  MoveL 3911 to (-68.86, -0.76, -116.32) mm, rotated rx -167.81 ry 3.47 rz -52.11 deg; joints [3.12, -29.463, 100.959, 149.35, 98.482, 24.468, -1.714]
  MoveL 3912 to (-69, -0.7, -116.34) mm, rotated rx -167.81 ry 3.47 rz -52.11 deg; joints [3.124, -29.466, 100.956, 149.354, 98.476, 24.47, -1.714]
  MoveL 3913 to (-69.11, -0.62, -116.37) mm, rotated rx -167.81 ry 3.47 rz -52.11 deg; joints [3.127, -29.469, 100.952, 149.358, 98.47, 24.473, -1.714]
  MoveL 3914 to (-69.19, -0.51, -116.39) mm, rotated rx -167.81 ry 3.47 rz -52.11 deg; joints [3.13, -29.471, 100.946, 149.36, 98.462, 24.477, -1.714]
  MoveL 3915 to (-69.26, -0.38, -116.42) mm, rotated rx -167.81 ry 3.47 rz -52.11 deg; joints [3.131, -29.473, 100.938, 149.362, 98.454, 24.481, -1.714]
  MoveL 3916 to (-69.34, -0.08, -116.48) mm, rotated rx -167.81 ry 3.47 rz -52.11 deg; joints [3.132, -29.476, 100.918, 149.365, 98.435, 24.492, -1.714]
  MoveL 3917 to (-69.29, 0.72, -116.61) mm, rotated rx -167.81 ry 3.47 rz -52.11 deg; joints [3.125, -29.476, 100.864, 149.363, 98.389, 24.522, -1.714]
  MoveL 3918 to (-69.03, 1.69, -116.75) mm, rotated rx -167.81 ry 3.47 rz -52.11 deg; joints [3.11, -29.47, 100.795, 149.353, 98.337, 24.559, -1.714]
  MoveL 3919 to (-68.14, 3.85, -117.02) mm, rotated rx -167.81 ry 3.47 rz -52.11 deg; joints [3.064, -29.451, 100.637, 149.322, 98.225, 24.643, -1.714]
  MoveL 3920 to (-67.07, 6.02, -117.26) mm, rotated rx -167.81 ry 3.47 rz -52.11 deg; joints [3.012, -29.425, 100.475, 149.285, 98.117, 24.728, -1.714]
  MoveL 3921 to (-42.84, 54.26, -122.35) mm, rotated rx -167.81 ry 3.47 rz -52.11 deg; joints [1.884, -28.742, 96.738, 148.461, 95.706, 26.658, -1.714]
  MoveL 3922 to (-41.12, 57.69, -122.71) mm, rotated rx -167.81 ry 3.47 rz -52.11 deg; joints [1.807, -28.687, 96.464, 148.402, 95.535, 26.798, -1.714]
  MoveL 3923 to (-39.28, 60.95, -123.12) mm, rotated rx -167.81 ry 3.47 rz -52.11 deg; joints [1.725, -28.634, 96.204, 148.34, 95.375, 26.934, -1.714]
  MoveL 3924 to (-38.32, 62.09, -123.33) mm, rotated rx -167.81 ry 3.47 rz -52.11 deg; joints [1.685, -28.614, 96.114, 148.307, 95.323, 26.984, -1.714]
  MoveL 3925 to (-37.87, 62.4, -123.43) mm, rotated rx -167.81 ry 3.47 rz -52.11 deg; joints [1.666, -28.607, 96.09, 148.292, 95.312, 26.999, -1.714]
  MoveL 3926 to (-37.65, 62.47, -123.47) mm, rotated rx -167.81 ry 3.47 rz -52.11 deg; joints [1.658, -28.605, 96.085, 148.284, 95.311, 27.004, -1.714]
  MoveL 3927 to (-37.44, 62.47, -123.52) mm, rotated rx -167.81 ry 3.47 rz -52.11 deg; joints [1.65, -28.604, 96.085, 148.277, 95.314, 27.006, -1.714]
  MoveL 3928 to (-37.25, 62.41, -123.55) mm, rotated rx -167.81 ry 3.47 rz -52.11 deg; joints [1.643, -28.603, 96.09, 148.271, 95.32, 27.005, -1.714]
  MoveL 3929 to (-37.06, 62.27, -123.59) mm, rotated rx -167.81 ry 3.47 rz -52.11 deg; joints [1.637, -28.604, 96.102, 148.264, 95.331, 27.001, -1.714]
  MoveL 3930 to (-36.88, 62.06, -123.62) mm, rotated rx -167.81 ry 3.47 rz -52.11 deg; joints [1.631, -28.606, 96.119, 148.258, 95.346, 26.995, -1.714]
  MoveL 3931 to (-36.72, 61.76, -123.64) mm, rotated rx -167.81 ry 3.47 rz -52.11 deg; joints [1.626, -28.609, 96.144, 148.253, 95.365, 26.985, -1.714]
  MoveL 3932 to (-36.22, 59.62, -123.69) mm, rotated rx -167.81 ry 3.47 rz -52.11 deg; joints [1.615, -28.632, 96.317, 148.236, 95.494, 26.909, -1.714]
  MoveL 3933 to (-35.96, 57.54, -123.69) mm, rotated rx -167.81 ry 3.47 rz -52.11 deg; joints [1.614, -28.656, 96.485, 148.227, 95.616, 26.834, -1.714]
  MoveL 3934 to (-35.96, 53.74, -123.74) mm, rotated rx -167.81 ry 3.47 rz -52.11 deg; joints [1.627, -28.711, 96.797, 148.225, 95.833, 26.693, -1.714]
  MoveL 3935 to (-36.73, 50.28, -123.85) mm, rotated rx -167.81 ry 3.47 rz -52.11 deg; joints [1.666, -28.779, 97.091, 148.248, 96.018, 26.561, -1.714]
  MoveL 3936 to (-39.45, 44.87, -124.14) mm, rotated rx -167.81 ry 3.47 rz -52.11 deg; joints [1.779, -28.918, 97.569, 148.33, 96.285, 26.346, -1.714]
  MoveL 3937 to (-40.92, 43.03, -124.27) mm, rotated rx -167.81 ry 3.47 rz -52.11 deg; joints [1.837, -28.977, 97.738, 148.376, 96.367, 26.27, -1.714]
  MoveL 3938 to (-63.78, 16.83, -126.14) mm, rotated rx -167.81 ry 3.47 rz -52.11 deg; joints [2.746, -29.822, 100.106, 149.099, 97.503, 25.201, -1.714]
  MoveL 3939 to (-65.73, 14.58, -126.3) mm, rotated rx -167.81 ry 3.47 rz -52.11 deg; joints [2.825, -29.892, 100.304, 149.161, 97.6, 25.111, -1.714]
  MoveL 3940 to (-67.81, 11.48, -126.54) mm, rotated rx -167.81 ry 3.47 rz -52.11 deg; joints [2.912, -29.978, 100.575, 149.227, 97.744, 24.99, -1.714]
  MoveL 3941 to (-68.34, 10.09, -126.68) mm, rotated rx -167.81 ry 3.47 rz -52.11 deg; joints [2.936, -30.011, 100.694, 149.243, 97.814, 24.939, -1.714]
  MoveL 3942 to (-68.38, 9.55, -126.75) mm, rotated rx -167.81 ry 3.47 rz -52.11 deg; joints [2.939, -30.022, 100.741, 149.243, 97.844, 24.92, -1.714]
  MoveL 3943 to (-68.32, 9.33, -126.79) mm, rotated rx -167.81 ry 3.47 rz -52.11 deg; joints [2.938, -30.025, 100.759, 149.241, 97.857, 24.912, -1.714]
  MoveL 3944 to (-68.22, 9.15, -126.83) mm, rotated rx -167.81 ry 3.47 rz -52.11 deg; joints [2.935, -30.028, 100.775, 149.237, 97.869, 24.906, -1.714]
  MoveL 3945 to (-68.07, 9.01, -126.86) mm, rotated rx -167.81 ry 3.47 rz -52.11 deg; joints [2.929, -30.029, 100.787, 149.231, 97.879, 24.902, -1.714]
  MoveL 3946 to (-67.85, 8.91, -126.9) mm, rotated rx -167.81 ry 3.47 rz -52.11 deg; joints [2.921, -30.028, 100.794, 149.223, 97.888, 24.9, -1.714]
  MoveL 3947 to (-67.58, 8.87, -126.93) mm, rotated rx -167.81 ry 3.47 rz -52.11 deg; joints [2.911, -30.025, 100.798, 149.214, 97.895, 24.9, -1.714]
  MoveL 3948 to (-67.23, 8.88, -126.96) mm, rotated rx -167.81 ry 3.47 rz -52.11 deg; joints [2.898, -30.021, 100.796, 149.202, 97.899, 24.902, -1.714]
  MoveL 3949 to (-65.14, 9.53, -127.09) mm, rotated rx -167.81 ry 3.47 rz -52.11 deg; joints [2.818, -29.984, 100.737, 149.13, 97.894, 24.937, -1.714]
  MoveL 3950 to (-64.67, 9.74, -127.11) mm, rotated rx -167.81 ry 3.47 rz -52.11 deg; joints [2.799, -29.975, 100.719, 149.114, 97.889, 24.947, -1.714]
  MoveL 3951 to (-64.25, 9.95, -127.15) mm, rotated rx -167.81 ry 3.47 rz -52.11 deg; joints [2.783, -29.968, 100.702, 149.1, 97.883, 24.957, -1.714]
  MoveL 3952 to (-63.87, 10.16, -127.23) mm, rotated rx -167.81 ry 3.47 rz -52.11 deg; joints [2.767, -29.964, 100.686, 149.087, 97.876, 24.967, -1.714]
  MoveL 3953 to (-63.48, 10.37, -127.28) mm, rotated rx -167.81 ry 3.47 rz -52.11 deg; joints [2.751, -29.958, 100.671, 149.073, 97.87, 24.977, -1.714]
  MoveL 3954 to (-63.06, 10.57, -127.32) mm, rotated rx -167.81 ry 3.47 rz -52.11 deg; joints [2.735, -29.951, 100.654, 149.059, 97.865, 24.986, -1.714]
  MoveL 3955 to (-58.72, 12.34, -127.33) mm, rotated rx -167.81 ry 3.47 rz -52.11 deg; joints [2.569, -29.854, 100.484, 148.914, 97.831, 25.072, -1.714]
  MoveL 3956 to (-58.31, 12.51, -127.35) mm, rotated rx -167.81 ry 3.47 rz -52.11 deg; joints [2.553, -29.846, 100.468, 148.9, 97.827, 25.08, -1.714]
  MoveL 3957 to (-57.88, 12.7, -127.36) mm, rotated rx -167.81 ry 3.47 rz -52.11 deg; joints [2.536, -29.836, 100.451, 148.886, 97.823, 25.089, -1.714]
  MoveL 3958 to (-56.92, 13.09, -127.36) mm, rotated rx -167.81 ry 3.47 rz -52.11 deg; joints [2.5, -29.815, 100.413, 148.854, 97.816, 25.108, -1.714]
  MoveL 3959 to (-56.39, 13.31, -127.37) mm, rotated rx -167.81 ry 3.47 rz -52.11 deg; joints [2.479, -29.803, 100.392, 148.836, 97.811, 25.119, -1.714]
  MoveL 3960 to (-55.85, 13.57, -127.39) mm, rotated rx -167.81 ry 3.47 rz -52.11 deg; joints [2.458, -29.792, 100.369, 148.818, 97.804, 25.131, -1.714]
  MoveL 3961 to (-55.26, 13.89, -127.42) mm, rotated rx -167.81 ry 3.47 rz -52.11 deg; joints [2.435, -29.78, 100.341, 148.798, 97.795, 25.146, -1.714]
  MoveL 3962 to (-54.72, 14.27, -127.44) mm, rotated rx -167.81 ry 3.47 rz -52.11 deg; joints [2.414, -29.767, 100.309, 148.78, 97.782, 25.163, -1.714]
  MoveL 3963 to (-54.22, 14.69, -127.45) mm, rotated rx -167.81 ry 3.47 rz -52.11 deg; joints [2.394, -29.754, 100.273, 148.764, 97.765, 25.181, -1.714]
  MoveL 3964 to (-55.39, 14.09, -128.43) mm, rotated rx -167.81 ry 3.47 rz -52.11 deg; joints [2.428, -29.845, 100.383, 148.793, 97.776, 25.161, -1.714]
  MoveL 3965 to (-54.92, 15.35, -128.86) mm, rotated rx -167.81 ry 3.47 rz -52.11 deg; joints [2.401, -29.85, 100.305, 148.775, 97.709, 25.212, -1.714]
  MoveL 3966 to (-54.28, 16.69, -129.18) mm, rotated rx -167.81 ry 3.47 rz -52.11 deg; joints [2.368, -29.844, 100.212, 148.751, 97.641, 25.267, -1.714]
  MoveL 3967 to (-53.45, 18.17, -129.41) mm, rotated rx -167.81 ry 3.47 rz -52.11 deg; joints [2.329, -29.828, 100.102, 148.723, 97.568, 25.327, -1.714]
  MoveL 3968 to (-52.29, 19.97, -129.63) mm, rotated rx -167.81 ry 3.47 rz -52.11 deg; joints [2.278, -29.801, 99.964, 148.683, 97.482, 25.4, -1.714]
  MoveL 3969 to (-51.11, 21.74, -129.75) mm, rotated rx -167.81 ry 3.47 rz -52.11 deg; joints [2.226, -29.767, 99.821, 148.645, 97.398, 25.472, -1.714]
  MoveL 3970 to (-49.93, 23.52, -129.86) mm, rotated rx -167.81 ry 3.47 rz -52.11 deg; joints [2.175, -29.732, 99.678, 148.606, 97.314, 25.545, -1.714]
  MoveL 3971 to (-48.77, 25.31, -130.09) mm, rotated rx -167.81 ry 3.47 rz -52.11 deg; joints [2.123, -29.705, 99.54, 148.566, 97.229, 25.618, -1.714]
  MoveL 3972 to (-47.58, 27.08, -130.2) mm, rotated rx -167.81 ry 3.47 rz -52.11 deg; joints [2.072, -29.67, 99.396, 148.527, 97.145, 25.691, -1.714]
  MoveL 3973 to (-46.4, 28.86, -130.44) mm, rotated rx -167.81 ry 3.47 rz -52.11 deg; joints [2.02, -29.643, 99.258, 148.488, 97.061, 25.764, -1.714]
  MoveL 3974 to (-45.21, 30.64, -130.55) mm, rotated rx -167.81 ry 3.47 rz -52.11 deg; joints [1.969, -29.608, 99.114, 148.449, 96.977, 25.837, -1.714]
  MoveL 3975 to (-44.02, 32.41, -130.67) mm, rotated rx -167.81 ry 3.47 rz -52.11 deg; joints [1.918, -29.572, 98.97, 148.41, 96.894, 25.91, -1.714]
  MoveL 3976 to (-42.83, 34.18, -130.91) mm, rotated rx -167.81 ry 3.47 rz -52.11 deg; joints [1.866, -29.544, 98.832, 148.37, 96.81, 25.984, -1.714]
  MoveL 3977 to (-41.68, 35.86, -131.01) mm, rotated rx -167.81 ry 3.47 rz -52.11 deg; joints [1.817, -29.509, 98.693, 148.332, 96.731, 26.053, -1.714]
  MoveL 3978 to (-40.55, 37.5, -131.22) mm, rotated rx -167.81 ry 3.47 rz -52.11 deg; joints [1.768, -29.481, 98.564, 148.294, 96.654, 26.122, -1.714]
  MoveL 3979 to (-39.23, 39.47, -131.38) mm, rotated rx -167.81 ry 3.47 rz -52.11 deg; joints [1.711, -29.443, 98.404, 148.251, 96.561, 26.204, -1.714]
  MoveL 3980 to (-37.68, 41.7, -131.47) mm, rotated rx -167.81 ry 3.47 rz -52.11 deg; joints [1.646, -29.391, 98.215, 148.201, 96.457, 26.296, -1.714]
  MoveL 3981 to (-36.51, 43.42, -131.53) mm, rotated rx -167.81 ry 3.47 rz -52.11 deg; joints [1.598, -29.352, 98.07, 148.164, 96.376, 26.367, -1.714]
  MoveL 3982 to (-35.43, 45.01, -131.66) mm, rotated rx -167.81 ry 3.47 rz -52.11 deg; joints [1.552, -29.32, 97.94, 148.128, 96.301, 26.434, -1.714]
  MoveL 3983 to (-34.31, 46.65, -131.76) mm, rotated rx -167.81 ry 3.47 rz -52.11 deg; joints [1.505, -29.285, 97.803, 148.092, 96.224, 26.502, -1.714]
  MoveL 3984 to (-33.21, 48.26, -131.88) mm, rotated rx -167.81 ry 3.47 rz -52.11 deg; joints [1.459, -29.25, 97.669, 148.056, 96.149, 26.57, -1.714]
  MoveL 3985 to (-32.04, 49.96, -131.95) mm, rotated rx -167.81 ry 3.47 rz -52.11 deg; joints [1.41, -29.211, 97.525, 148.019, 96.069, 26.641, -1.714]
  MoveL 3986 to (-30.78, 51.79, -132.04) mm, rotated rx -167.81 ry 3.47 rz -52.11 deg; joints [1.358, -29.169, 97.37, 147.978, 95.983, 26.718, -1.714]
  MoveL 3987 to (-29.39, 53.75, -132.31) mm, rotated rx -167.81 ry 3.47 rz -52.11 deg; joints [1.299, -29.133, 97.212, 147.932, 95.891, 26.802, -1.714]
  MoveL 3988 to (-28.56, 55.83, -133.29) mm, rotated rx -167.81 ry 3.47 rz -52.11 deg; joints [1.251, -29.152, 97.089, 147.897, 95.781, 26.893, -1.714]
  MoveL 3989 to (-28.58, 54.69, -133.78) mm, rotated rx -167.81 ry 3.47 rz -52.11 deg; joints [1.25, -29.199, 97.209, 147.892, 95.843, 26.854, -1.714]
  MoveL 3990 to (-28.58, 54.09, -134.09) mm, rotated rx -167.81 ry 3.47 rz -52.11 deg; joints [1.249, -29.227, 97.275, 147.889, 95.875, 26.834, -1.714]
  MoveL 3991 to (-28.58, 54, -134.24) mm, rotated rx -167.81 ry 3.47 rz -52.11 deg; joints [1.248, -29.238, 97.291, 147.888, 95.88, 26.832, -1.714]
  MoveL 3992 to (-28.57, 54.34, -134.27) mm, rotated rx -167.81 ry 3.47 rz -52.11 deg; joints [1.246, -29.235, 97.265, 147.887, 95.861, 26.845, -1.714]
  MoveL 3993 to (-28.56, 54.81, -134.29) mm, rotated rx -167.81 ry 3.47 rz -52.11 deg; joints [1.244, -29.23, 97.228, 147.887, 95.834, 26.862, -1.714]
  MoveL 3994 to (-28.54, 55.29, -134.32) mm, rotated rx -167.81 ry 3.47 rz -52.11 deg; joints [1.241, -29.225, 97.19, 147.886, 95.807, 26.881, -1.714]
  MoveL 3995 to (-28.5, 55.74, -134.38) mm, rotated rx -167.81 ry 3.47 rz -52.11 deg; joints [1.237, -29.222, 97.157, 147.885, 95.782, 26.898, -1.714]
  MoveL 3996 to (-28.47, 56.2, -134.43) mm, rotated rx -167.81 ry 3.47 rz -52.11 deg; joints [1.234, -29.218, 97.121, 147.884, 95.756, 26.916, -1.714]
  MoveL 3997 to (-28.46, 56.69, -134.44) mm, rotated rx -167.81 ry 3.47 rz -52.11 deg; joints [1.232, -29.212, 97.082, 147.884, 95.728, 26.934, -1.714]
  MoveL 3998 to (-28.45, 59.31, -134.44) mm, rotated rx -167.81 ry 3.47 rz -52.11 deg; joints [1.223, -29.175, 96.868, 147.885, 95.58, 27.032, -1.714]
  MoveL 3999 to (-28.43, 59.76, -134.46) mm, rotated rx -167.81 ry 3.47 rz -52.11 deg; joints [1.22, -29.17, 96.832, 147.884, 95.554, 27.05, -1.714]
  MoveL 4000 to (-28.4, 60.15, -134.5) mm, rotated rx -167.81 ry 3.47 rz -52.11 deg; joints [1.218, -29.166, 96.802, 147.883, 95.532, 27.064, -1.714]
  MoveL 4001 to (-28.39, 60.61, -134.52) mm, rotated rx -167.81 ry 3.47 rz -52.11 deg; joints [1.215, -29.161, 96.765, 147.883, 95.506, 27.082, -1.714]
  MoveL 4002 to (-28.37, 61.21, -134.54) mm, rotated rx -167.81 ry 3.47 rz -52.11 deg; joints [1.213, -29.153, 96.717, 147.882, 95.473, 27.104, -1.714]
  MoveL 4003 to (-28.33, 61.93, -134.6) mm, rotated rx -167.81 ry 3.47 rz -52.11 deg; joints [1.208, -29.146, 96.66, 147.881, 95.432, 27.132, -1.714]
  MoveL 4004 to (-28.31, 62.55, -134.62) mm, rotated rx -167.81 ry 3.47 rz -52.11 deg; joints [1.205, -29.138, 96.611, 147.88, 95.397, 27.156, -1.714]
  MoveL 4005 to (-28.3, 63.08, -134.63) mm, rotated rx -167.81 ry 3.47 rz -52.11 deg; joints [1.203, -29.131, 96.568, 147.88, 95.367, 27.175, -1.714]
  MoveL 4006 to (-28.29, 64.65, -134.63) mm, rotated rx -167.81 ry 3.47 rz -52.11 deg; joints [1.197, -29.108, 96.438, 147.88, 95.278, 27.234, -1.714]
  MoveL 4007 to (-27.99, 67.55, -134.97) mm, rotated rx -167.81 ry 3.47 rz -52.11 deg; joints [1.173, -29.082, 96.216, 147.868, 95.116, 27.347, -1.714]
  MoveL 4008 to (-27.61, 68.79, -135.4) mm, rotated rx -167.81 ry 3.47 rz -52.11 deg; joints [1.151, -29.084, 96.133, 147.852, 95.049, 27.4, -1.714]
  MoveL 4009 to (-27.09, 69.89, -136) mm, rotated rx -167.81 ry 3.47 rz -52.11 deg; joints [1.122, -29.096, 96.07, 147.83, 94.992, 27.449, -1.714]
  MoveL 4010 to (-25.61, 71.68, -137.71) mm, rotated rx -167.81 ry 3.47 rz -52.11 deg; joints [1.046, -29.15, 96.002, 147.768, 94.904, 27.54, -1.714]
  MoveL 4011 to (-23.55, 72.91, -140.1) mm, rotated rx -167.81 ry 3.47 rz -52.11 deg; joints [0.942, -29.245, 96.011, 147.679, 94.854, 27.62, -1.714]
  MoveL 4012 to (-21.54, 73.36, -142.5) mm, rotated rx -167.81 ry 3.47 rz -52.11 deg; joints [0.844, -29.352, 96.085, 147.593, 94.847, 27.671, -1.714]
  MoveL 4013 to (-20.79, 73.19, -143.44) mm, rotated rx -167.81 ry 3.47 rz -52.11 deg; joints [0.807, -29.4, 96.143, 147.56, 94.863, 27.678, -1.714]
  MoveL 4014 to (-20.22, 72.77, -144.21) mm, rotated rx -167.81 ry 3.47 rz -52.11 deg; joints [0.78, -29.444, 96.214, 147.535, 94.891, 27.673, -1.714]
  MoveL 4015 to (-20, 72.47, -144.53) mm, rotated rx -167.81 ry 3.47 rz -52.11 deg; joints [0.77, -29.465, 96.255, 147.525, 94.91, 27.666, -1.714]
  MoveL 4016 to (-19.82, 72.1, -144.81) mm, rotated rx -167.81 ry 3.47 rz -52.11 deg; joints [0.761, -29.485, 96.299, 147.516, 94.932, 27.655, -1.714]
  MoveL 4017 to (-19.6, 71.17, -145.24) mm, rotated rx -167.81 ry 3.47 rz -52.11 deg; joints [0.752, -29.522, 96.397, 147.505, 94.986, 27.625, -1.714]
  MoveL 4018 to (-19.54, 69.98, -145.49) mm, rotated rx -167.81 ry 3.47 rz -52.11 deg; joints [0.751, -29.555, 96.509, 147.5, 95.053, 27.583, -1.714]
  MoveL 4019 to (-19.67, 68.53, -145.58) mm, rotated rx -167.81 ry 3.47 rz -52.11 deg; joints [0.758, -29.584, 96.634, 147.502, 95.132, 27.529, -1.714]
  MoveL 4020 to (-19.74, 68.01, -145.58) mm, rotated rx -167.81 ry 3.47 rz -52.11 deg; joints [0.762, -29.593, 96.677, 147.504, 95.161, 27.509, -1.714]
  MoveL 4021 to (-19.83, 67.58, -145.52) mm, rotated rx -167.81 ry 3.47 rz -52.11 deg; joints [0.768, -29.597, 96.711, 147.508, 95.184, 27.492, -1.714]
  MoveL 4022 to (-19.93, 67.16, -145.46) mm, rotated rx -167.81 ry 3.47 rz -52.11 deg; joints [0.773, -29.602, 96.743, 147.511, 95.206, 27.474, -1.714]
  MoveL 4023 to (-20.02, 66.69, -145.43) mm, rotated rx -167.81 ry 3.47 rz -52.11 deg; joints [0.778, -29.608, 96.781, 147.514, 95.232, 27.456, -1.714]
  MoveL 4024 to (-20.1, 66.2, -145.41) mm, rotated rx -167.81 ry 3.47 rz -52.11 deg; joints [0.783, -29.615, 96.821, 147.516, 95.258, 27.437, -1.714]
  MoveL 4025 to (-20.17, 65.68, -145.4) mm, rotated rx -167.81 ry 3.47 rz -52.11 deg; joints [0.787, -29.624, 96.865, 147.518, 95.287, 27.417, -1.714]
  MoveL 4026 to (-20.24, 65.16, -145.4) mm, rotated rx -167.81 ry 3.47 rz -52.11 deg; joints [0.791, -29.633, 96.908, 147.52, 95.315, 27.397, -1.714]
  MoveL 4027 to (-20.3, 64.65, -145.42) mm, rotated rx -167.81 ry 3.47 rz -52.11 deg; joints [0.794, -29.642, 96.951, 147.522, 95.343, 27.377, -1.714]
  MoveL 4028 to (-20.35, 64.16, -145.43) mm, rotated rx -167.81 ry 3.47 rz -52.11 deg; joints [0.798, -29.651, 96.993, 147.523, 95.37, 27.359, -1.714]
  MoveL 4029 to (-20.42, 63.7, -145.41) mm, rotated rx -167.81 ry 3.47 rz -52.11 deg; joints [0.802, -29.657, 97.03, 147.525, 95.395, 27.341, -1.714]
  MoveL 4030 to (-20.51, 63.24, -145.37) mm, rotated rx -167.81 ry 3.47 rz -52.11 deg; joints [0.807, -29.663, 97.066, 147.528, 95.42, 27.323, -1.714]
  MoveL 4031 to (-20.61, 62.71, -145.32) mm, rotated rx -167.81 ry 3.47 rz -52.11 deg; joints [0.813, -29.669, 97.108, 147.531, 95.449, 27.301, -1.714]
  MoveL 4032 to (-20.75, 62.02, -145.27) mm, rotated rx -167.81 ry 3.47 rz -52.11 deg; joints [0.82, -29.679, 97.163, 147.536, 95.486, 27.274, -1.714]
  MoveL 4033 to (-20.86, 61.38, -145.24) mm, rotated rx -167.81 ry 3.47 rz -52.11 deg; joints [0.826, -29.688, 97.215, 147.539, 95.52, 27.249, -1.714]
  MoveL 4034 to (-21.2, 58.79, -145.24) mm, rotated rx -167.81 ry 3.47 rz -52.11 deg; joints [0.847, -29.731, 97.431, 147.548, 95.662, 27.15, -1.714]
  MoveL 4035 to (-21.3, 58.17, -145.21) mm, rotated rx -167.81 ry 3.47 rz -52.11 deg; joints [0.853, -29.739, 97.48, 147.551, 95.696, 27.126, -1.714]
  MoveL 4036 to (-21.4, 57.62, -145.15) mm, rotated rx -167.81 ry 3.47 rz -52.11 deg; joints [0.859, -29.745, 97.523, 147.555, 95.725, 27.104, -1.714]
  MoveL 4037 to (-21.44, 57.42, -145) mm, rotated rx -167.81 ry 3.47 rz -52.11 deg; joints [0.862, -29.739, 97.532, 147.557, 95.737, 27.095, -1.714]
  MoveL 4038 to (-21.42, 57.54, -144.73) mm, rotated rx -167.81 ry 3.47 rz -52.11 deg; joints [0.864, -29.72, 97.507, 147.559, 95.732, 27.097, -1.714]
  MoveL 4039 to (-21.33, 57.99, -144.33) mm, rotated rx -167.81 ry 3.47 rz -52.11 deg; joints [0.864, -29.687, 97.448, 147.56, 95.71, 27.111, -1.714]
  MoveL 4040 to (-22.34, 57.8, -143.53) mm, rotated rx -167.81 ry 3.47 rz -52.11 deg; joints [0.91, -29.658, 97.43, 147.601, 95.71, 27.09, -1.714]
  MoveL 4041 to (-23.69, 56.35, -143.31) mm, rotated rx -167.81 ry 3.47 rz -52.11 deg; joints [0.965, -29.689, 97.549, 147.645, 95.773, 27.025, -1.714]
  MoveL 4042 to (-25.04, 54.87, -143.15) mm, rotated rx -167.81 ry 3.47 rz -52.11 deg; joints [1.019, -29.725, 97.674, 147.689, 95.838, 26.96, -1.714]
  MoveL 4043 to (-26.42, 53.34, -143) mm, rotated rx -167.81 ry 3.47 rz -52.11 deg; joints [1.075, -29.762, 97.803, 147.734, 95.905, 26.893, -1.714]
  MoveL 4044 to (-27.69, 51.96, -142.71) mm, rotated rx -167.81 ry 3.47 rz -52.11 deg; joints [1.128, -29.786, 97.912, 147.777, 95.966, 26.83, -1.714]
  MoveL 4045 to (-29.11, 50.39, -142.52) mm, rotated rx -167.81 ry 3.47 rz -52.11 deg; joints [1.186, -29.821, 98.042, 147.823, 96.034, 26.761, -1.714]
  MoveL 4046 to (-30.59, 48.75, -142.33) mm, rotated rx -167.81 ry 3.47 rz -52.11 deg; joints [1.247, -29.859, 98.179, 147.872, 96.106, 26.689, -1.714]
  MoveL 4047 to (-32.09, 47.08, -142.25) mm, rotated rx -167.81 ry 3.47 rz -52.11 deg; joints [1.307, -29.903, 98.323, 147.92, 96.179, 26.617, -1.714]
  MoveL 4048 to (-33.9, 45.04, -142.16) mm, rotated rx -167.81 ry 3.47 rz -52.11 deg; joints [1.38, -29.958, 98.499, 147.979, 96.268, 26.529, -1.714]
  MoveL 4049 to (-35.2, 43.57, -142.05) mm, rotated rx -167.81 ry 3.47 rz -52.11 deg; joints [1.433, -29.994, 98.623, 148.021, 96.332, 26.466, -1.714]
  MoveL 4050 to (-36.41, 42.2, -141.83) mm, rotated rx -167.81 ry 3.47 rz -52.11 deg; joints [1.483, -30.021, 98.732, 148.061, 96.392, 26.406, -1.714]
  MoveL 4051 to (-37.75, 40.69, -141.64) mm, rotated rx -167.81 ry 3.47 rz -52.11 deg; joints [1.539, -30.053, 98.855, 148.106, 96.459, 26.341, -1.714]
  MoveL 4052 to (-39.16, 39.09, -141.52) mm, rotated rx -167.81 ry 3.47 rz -52.11 deg; joints [1.597, -30.091, 98.99, 148.152, 96.529, 26.272, -1.714]
  MoveL 4053 to (-40.55, 37.5, -141.35) mm, rotated rx -167.81 ry 3.47 rz -52.11 deg; joints [1.654, -30.126, 99.12, 148.198, 96.6, 26.204, -1.714]
  MoveL 4054 to (-41.94, 35.91, -141.23) mm, rotated rx -167.81 ry 3.47 rz -52.11 deg; joints [1.712, -30.163, 99.252, 148.244, 96.669, 26.136, -1.714]
  MoveL 4055 to (-43.37, 34.26, -141.05) mm, rotated rx -167.81 ry 3.47 rz -52.11 deg; joints [1.771, -30.199, 99.386, 148.291, 96.742, 26.066, -1.714]
  MoveL 4056 to (-44.77, 32.65, -140.93) mm, rotated rx -167.81 ry 3.47 rz -52.11 deg; joints [1.829, -30.236, 99.519, 148.337, 96.813, 25.997, -1.714]
  MoveL 4057 to (-46.15, 31.03, -140.7) mm, rotated rx -167.81 ry 3.47 rz -52.11 deg; joints [1.888, -30.267, 99.648, 148.384, 96.885, 25.928, -1.714]
  MoveL 4058 to (-47.55, 29.41, -140.58) mm, rotated rx -167.81 ry 3.47 rz -52.11 deg; joints [1.946, -30.305, 99.781, 148.43, 96.956, 25.86, -1.714]
  MoveL 4059 to (-48.94, 27.8, -140.47) mm, rotated rx -167.81 ry 3.47 rz -52.11 deg; joints [2.004, -30.342, 99.914, 148.476, 97.027, 25.792, -1.714]
  MoveL 4060 to (-50.32, 26.16, -140.24) mm, rotated rx -167.81 ry 3.47 rz -52.11 deg; joints [2.063, -30.372, 100.043, 148.523, 97.1, 25.722, -1.714]
  MoveL 4061 to (-51.53, 24.65, -140.04) mm, rotated rx -167.81 ry 3.47 rz -52.11 deg; joints [2.115, -30.399, 100.161, 148.564, 97.168, 25.659, -1.714]
  MoveL 4062 to (-52.58, 23.23, -139.75) mm, rotated rx -167.81 ry 3.47 rz -52.11 deg; joints [2.162, -30.416, 100.265, 148.6, 97.234, 25.599, -1.714]
  MoveL 4063 to (-53.49, 21.88, -139.34) mm, rotated rx -167.81 ry 3.47 rz -52.11 deg; joints [2.205, -30.422, 100.357, 148.633, 97.3, 25.541, -1.714]
  MoveL 4064 to (-52.18, 22.58, -138.42) mm, rotated rx -167.81 ry 3.47 rz -52.11 deg; joints [2.165, -30.331, 100.241, 148.599, 97.286, 25.566, -1.714]
  MoveL 4065 to (-52.64, 22.23, -138.41) mm, rotated rx -167.81 ry 3.47 rz -52.11 deg; joints [2.183, -30.343, 100.271, 148.614, 97.298, 25.551, -1.714]
  MoveL 4066 to (-53.09, 21.94, -138.38) mm, rotated rx -167.81 ry 3.47 rz -52.11 deg; joints [2.201, -30.353, 100.296, 148.629, 97.308, 25.538, -1.714]
  MoveL 4067 to (-53.5, 21.72, -138.32) mm, rotated rx -167.81 ry 3.47 rz -52.11 deg; joints [2.217, -30.359, 100.313, 148.643, 97.314, 25.527, -1.714]
  MoveL 4068 to (-53.91, 21.54, -138.26) mm, rotated rx -167.81 ry 3.47 rz -52.11 deg; joints [2.234, -30.364, 100.328, 148.657, 97.319, 25.518, -1.714]
  MoveL 4069 to (-54.34, 21.38, -138.21) mm, rotated rx -167.81 ry 3.47 rz -52.11 deg; joints [2.251, -30.371, 100.341, 148.672, 97.322, 25.509, -1.714]
  MoveL 4070 to (-54.81, 21.23, -138.17) mm, rotated rx -167.81 ry 3.47 rz -52.11 deg; joints [2.268, -30.379, 100.355, 148.688, 97.324, 25.501, -1.714]
  MoveL 4071 to (-55.31, 21.08, -138.16) mm, rotated rx -167.81 ry 3.47 rz -52.11 deg; joints [2.288, -30.389, 100.369, 148.705, 97.324, 25.493, -1.714]
  MoveL 4072 to (-55.82, 20.95, -138.16) mm, rotated rx -167.81 ry 3.47 rz -52.11 deg; joints [2.307, -30.4, 100.384, 148.722, 97.324, 25.486, -1.714]
  MoveL 4073 to (-56.27, 20.82, -138.15) mm, rotated rx -167.81 ry 3.47 rz -52.11 deg; joints [2.324, -30.409, 100.397, 148.737, 97.324, 25.478, -1.714]
  MoveL 4074 to (-56.67, 20.69, -138.12) mm, rotated rx -167.81 ry 3.47 rz -52.11 deg; joints [2.339, -30.416, 100.409, 148.75, 97.326, 25.471, -1.714]
  MoveL 4075 to (-57.14, 20.55, -138.11) mm, rotated rx -167.81 ry 3.47 rz -52.11 deg; joints [2.357, -30.425, 100.422, 148.766, 97.326, 25.464, -1.714]
  MoveL 4076 to (-57.64, 20.42, -138.11) mm, rotated rx -167.81 ry 3.47 rz -52.11 deg; joints [2.375, -30.436, 100.437, 148.783, 97.326, 25.457, -1.714]
  MoveL 4077 to (-58.23, 20.25, -138.09) mm, rotated rx -167.81 ry 3.47 rz -52.11 deg; joints [2.398, -30.447, 100.453, 148.803, 97.327, 25.447, -1.714]
  MoveL 4078 to (-58.9, 20.05, -138.04) mm, rotated rx -167.81 ry 3.47 rz -52.11 deg; joints [2.423, -30.459, 100.471, 148.825, 97.328, 25.436, -1.714]
  MoveL 4079 to (-59.48, 19.89, -138.02) mm, rotated rx -167.81 ry 3.47 rz -52.11 deg; joints [2.445, -30.47, 100.488, 148.845, 97.328, 25.427, -1.714]
  MoveL 4080 to (-60.1, 19.71, -138) mm, rotated rx -167.81 ry 3.47 rz -52.11 deg; joints [2.469, -30.482, 100.505, 148.865, 97.329, 25.417, -1.714]
  MoveL 4081 to (-60.78, 19.49, -137.96) mm, rotated rx -167.81 ry 3.47 rz -52.11 deg; joints [2.495, -30.494, 100.525, 148.888, 97.331, 25.406, -1.714]
  MoveL 4082 to (-61.34, 19.33, -137.95) mm, rotated rx -167.81 ry 3.47 rz -52.11 deg; joints [2.516, -30.505, 100.541, 148.907, 97.331, 25.397, -1.714]
  MoveL 4083 to (-61.87, 19.19, -137.94) mm, rotated rx -167.81 ry 3.47 rz -52.11 deg; joints [2.536, -30.516, 100.556, 148.925, 97.331, 25.389, -1.714]
  MoveL 4084 to (-63.39, 18.79, -137.94) mm, rotated rx -167.81 ry 3.47 rz -52.11 deg; joints [2.593, -30.548, 100.599, 148.976, 97.33, 25.367, -1.714]
  MoveL 4085 to (-64.81, 18.49, -138.03) mm, rotated rx -167.81 ry 3.47 rz -52.11 deg; joints [2.645, -30.583, 100.637, 149.022, 97.324, 25.349, -1.714]
  MoveL 4086 to (-65.99, 18.39, -138.28) mm, rotated rx -167.81 ry 3.47 rz -52.11 deg; joints [2.686, -30.622, 100.667, 149.06, 97.31, 25.342, -1.714]
  MoveL 4087 to (-66.95, 18.5, -138.7) mm, rotated rx -167.81 ry 3.47 rz -52.11 deg; joints [2.715, -30.665, 100.689, 149.088, 97.286, 25.344, -1.714]
  MoveL 4088 to (-67.33, 18.63, -138.98) mm, rotated rx -167.81 ry 3.47 rz -52.11 deg; joints [2.726, -30.688, 100.696, 149.098, 97.271, 25.349, -1.714]
  MoveL 4089 to (-67.66, 18.81, -139.29) mm, rotated rx -167.81 ry 3.47 rz -52.11 deg; joints [2.733, -30.712, 100.702, 149.106, 97.253, 25.357, -1.714]
  MoveL 4090 to (-68.15, 19.32, -140.05) mm, rotated rx -167.81 ry 3.47 rz -52.11 deg; joints [2.74, -30.764, 100.706, 149.116, 97.212, 25.379, -1.714]
  MoveL 4091 to (-68.4, 20.04, -140.98) mm, rotated rx -167.81 ry 3.47 rz -52.11 deg; joints [2.736, -30.819, 100.702, 149.116, 97.161, 25.411, -1.714]
  MoveL 4092 to (-68.2, 22.08, -143.34) mm, rotated rx -167.81 ry 3.47 rz -52.11 deg; joints [2.694, -30.943, 100.668, 149.088, 97.033, 25.506, -1.714]
  MoveL 4093 to (-67.23, 24.28, -145.71) mm, rotated rx -167.81 ry 3.47 rz -52.11 deg; joints [2.623, -31.051, 100.615, 149.034, 96.908, 25.61, -1.714]
  MoveL 4094 to (-65.63, 25.97, -147.39) mm, rotated rx -167.81 ry 3.47 rz -52.11 deg; joints [2.539, -31.11, 100.562, 148.965, 96.827, 25.694, -1.714]
  MoveL 4095 to (-64.6, 26.62, -147.98) mm, rotated rx -167.81 ry 3.47 rz -52.11 deg; joints [2.492, -31.122, 100.535, 148.925, 96.802, 25.728, -1.714]
  MoveL 4096 to (-63.41, 27.14, -148.41) mm, rotated rx -167.81 ry 3.47 rz -52.11 deg; joints [2.442, -31.121, 100.507, 148.882, 96.789, 25.757, -1.714]
  MoveL 4097 to (-60.57, 27.81, -148.74) mm, rotated rx -167.81 ry 3.47 rz -52.11 deg; joints [2.333, -31.083, 100.452, 148.785, 96.794, 25.799, -1.714]
  MoveL 4098 to (-56.42, 28.35, -148.74) mm, rotated rx -167.81 ry 3.47 rz -52.11 deg; joints [2.18, -31, 100.378, 148.647, 96.829, 25.841, -1.714]
  MoveL 4099 to (-55.88, 28.43, -148.76) mm, rotated rx -167.81 ry 3.47 rz -52.11 deg; joints [2.16, -30.991, 100.368, 148.629, 96.832, 25.847, -1.714]
  MoveL 4100 to (-55.36, 28.53, -148.8) mm, rotated rx -167.81 ry 3.47 rz -52.11 deg; joints [2.14, -30.983, 100.359, 148.611, 96.835, 25.854, -1.714]
  MoveL 4101 to (-54.84, 28.64, -148.86) mm, rotated rx -167.81 ry 3.47 rz -52.11 deg; joints [2.12, -30.976, 100.349, 148.593, 96.836, 25.861, -1.714]
  MoveL 4102 to (-54.34, 28.76, -148.95) mm, rotated rx -167.81 ry 3.47 rz -52.11 deg; joints [2.101, -30.97, 100.34, 148.576, 96.836, 25.869, -1.714]
  MoveL 4103 to (-53.84, 28.88, -149.02) mm, rotated rx -167.81 ry 3.47 rz -52.11 deg; joints [2.081, -30.965, 100.331, 148.559, 96.837, 25.877, -1.714]
  MoveL 4104 to (-53.37, 28.97, -149.06) mm, rotated rx -167.81 ry 3.47 rz -52.11 deg; joints [2.063, -30.958, 100.322, 148.543, 96.839, 25.883, -1.714]
  MoveL 4105 to (-52.89, 29.04, -149.08) mm, rotated rx -167.81 ry 3.47 rz -52.11 deg; joints [2.046, -30.949, 100.314, 148.527, 96.842, 25.889, -1.714]
  MoveL 4106 to (-52.37, 29.11, -149.08) mm, rotated rx -167.81 ry 3.47 rz -52.11 deg; joints [2.027, -30.939, 100.304, 148.509, 96.846, 25.894, -1.714]
  MoveL 4107 to (-51.75, 29.21, -149.11) mm, rotated rx -167.81 ry 3.47 rz -52.11 deg; joints [2.003, -30.928, 100.293, 148.489, 96.85, 25.901, -1.714]
  MoveL 4108 to (-51.08, 29.34, -149.17) mm, rotated rx -167.81 ry 3.47 rz -52.11 deg; joints [1.978, -30.918, 100.281, 148.466, 96.853, 25.91, -1.714]
  MoveL 4109 to (-50.5, 29.45, -149.19) mm, rotated rx -167.81 ry 3.47 rz -52.11 deg; joints [1.956, -30.907, 100.268, 148.446, 96.855, 25.918, -1.714]
  MoveL 4110 to (-49.96, 29.6, -149.2) mm, rotated rx -167.81 ry 3.47 rz -52.11 deg; joints [1.936, -30.896, 100.253, 148.429, 96.855, 25.926, -1.714]
  MoveL 4111 to (-49.44, 29.79, -149.21) mm, rotated rx -167.81 ry 3.47 rz -52.11 deg; joints [1.916, -30.885, 100.233, 148.412, 96.853, 25.936, -1.714]
  MoveL 4112 to (-48.96, 30.1, -149.21) mm, rotated rx -167.81 ry 3.47 rz -52.11 deg; joints [1.898, -30.872, 100.205, 148.396, 96.843, 25.95, -1.714]
  MoveL 4113 to (-48.48, 30.48, -149.21) mm, rotated rx -167.81 ry 3.47 rz -52.11 deg; joints [1.879, -30.859, 100.171, 148.38, 96.828, 25.967, -1.714]
  MoveL 4114 to (-49.9, 29.8, -150.16) mm, rotated rx -167.81 ry 3.47 rz -52.11 deg; joints [1.922, -30.954, 100.288, 148.418, 96.839, 25.942, -1.714]
  MoveL 4115 to (-49.13, 30.78, -150.59) mm, rotated rx -167.81 ry 3.47 rz -52.11 deg; joints [1.886, -30.955, 100.227, 148.389, 96.793, 25.986, -1.714]
  MoveL 4116 to (-48.17, 31.82, -150.91) mm, rotated rx -167.81 ry 3.47 rz -52.11 deg; joints [1.844, -30.945, 100.153, 148.355, 96.746, 26.033, -1.714]
  MoveL 4117 to (-47.03, 32.96, -151.16) mm, rotated rx -167.81 ry 3.47 rz -52.11 deg; joints [1.795, -30.926, 100.067, 148.315, 96.698, 26.083, -1.714]
  MoveL 4118 to (-45.45, 34.38, -151.27) mm, rotated rx -167.81 ry 3.47 rz -52.11 deg; joints [1.731, -30.887, 99.947, 148.263, 96.641, 26.145, -1.714]
  MoveL 4119 to (-43.87, 35.82, -151.5) mm, rotated rx -167.81 ry 3.47 rz -52.11 deg; joints [1.666, -30.854, 99.831, 148.21, 96.583, 26.209, -1.714]
  MoveL 4120 to (-42.28, 37.24, -151.62) mm, rotated rx -167.81 ry 3.47 rz -52.11 deg; joints [1.603, -30.814, 99.711, 148.157, 96.526, 26.271, -1.714]
  MoveL 4121 to (-40.69, 38.65, -151.74) mm, rotated rx -167.81 ry 3.47 rz -52.11 deg; joints [1.539, -30.774, 99.59, 148.105, 96.47, 26.334, -1.714]
  MoveL 4122 to (-39.1, 40.08, -151.97) mm, rotated rx -167.81 ry 3.47 rz -52.11 deg; joints [1.474, -30.742, 99.474, 148.051, 96.412, 26.398, -1.714]
  MoveL 4123 to (-37.5, 41.49, -152.09) mm, rotated rx -167.81 ry 3.47 rz -52.11 deg; joints [1.41, -30.702, 99.353, 147.999, 96.356, 26.461, -1.714]
  MoveL 4124 to (-35.9, 42.9, -152.21) mm, rotated rx -167.81 ry 3.47 rz -52.11 deg; joints [1.346, -30.661, 99.232, 147.947, 96.3, 26.524, -1.714]
  MoveL 4125 to (-34.06, 44.53, -152.37) mm, rotated rx -167.81 ry 3.47 rz -52.11 deg; joints [1.273, -30.616, 99.093, 147.886, 96.234, 26.597, -1.714]
  MoveL 4126 to (-32.48, 45.92, -152.56) mm, rotated rx -167.81 ry 3.47 rz -52.11 deg; joints [1.209, -30.581, 98.978, 147.834, 96.179, 26.66, -1.714]
  MoveL 4127 to (-30.75, 47.44, -152.76) mm, rotated rx -167.81 ry 3.47 rz -52.11 deg; joints [1.139, -30.541, 98.849, 147.776, 96.118, 26.729, -1.714]
  MoveL 4128 to (-29.04, 48.92, -153.01) mm, rotated rx -167.81 ry 3.47 rz -52.11 deg; joints [1.071, -30.505, 98.727, 147.72, 96.058, 26.797, -1.714]
  MoveL 4129 to (-27.43, 50.33, -153.14) mm, rotated rx -167.81 ry 3.47 rz -52.11 deg; joints [1.007, -30.464, 98.605, 147.667, 96.003, 26.861, -1.714]
  MoveL 4130 to (-25.83, 51.73, -153.14) mm, rotated rx -167.81 ry 3.47 rz -52.11 deg; joints [0.945, -30.415, 98.476, 147.616, 95.947, 26.923, -1.714]
  MoveL 4131 to (-24.24, 53.11, -153.21) mm, rotated rx -167.81 ry 3.47 rz -52.11 deg; joints [0.883, -30.371, 98.353, 147.565, 95.893, 26.986, -1.714]
  MoveL 4132 to (-22.67, 54.45, -153.43) mm, rotated rx -167.81 ry 3.47 rz -52.11 deg; joints [0.82, -30.337, 98.241, 147.514, 95.84, 27.048, -1.714]
  MoveL 4133 to (-20.9, 55.92, -153.78) mm, rotated rx -167.81 ry 3.47 rz -52.11 deg; joints [0.749, -30.305, 98.122, 147.454, 95.781, 27.118, -1.714]
  MoveL 4134 to (-19.51, 57.08, -153.99) mm, rotated rx -167.81 ry 3.47 rz -52.11 deg; joints [0.693, -30.276, 98.025, 147.409, 95.735, 27.172, -1.714]
  MoveL 4135 to (-17.61, 58.64, -154.29) mm, rotated rx -167.81 ry 3.47 rz -52.11 deg; joints [0.618, -30.238, 97.895, 147.346, 95.673, 27.246, -1.714]
  MoveL 4136 to (-15.93, 60.07, -154.39) mm, rotated rx -167.81 ry 3.47 rz -52.11 deg; joints [0.553, -30.192, 97.767, 147.292, 95.617, 27.312, -1.714]
  MoveL 4137 to (-14.33, 61.47, -154.41) mm, rotated rx -167.81 ry 3.47 rz -52.11 deg; joints [0.491, -30.143, 97.637, 147.242, 95.561, 27.376, -1.714]
  MoveL 4138 to (-13.45, 61.58, -155.19) mm, rotated rx -167.81 ry 3.47 rz -52.11 deg; joints [0.451, -30.174, 97.66, 147.206, 95.564, 27.393, -1.714]
  MoveL 4139 to (-13.64, 61.18, -155.59) mm, rotated rx -167.81 ry 3.47 rz -52.11 deg; joints [0.454, -30.208, 97.716, 147.208, 95.581, 27.38, -1.714]
  MoveL 4140 to (-13.71, 61.06, -155.83) mm, rotated rx -167.81 ry 3.47 rz -52.11 deg; joints [0.454, -30.227, 97.74, 147.208, 95.585, 27.377, -1.714]
  MoveL 4141 to (-13.67, 61.2, -155.95) mm, rotated rx -167.81 ry 3.47 rz -52.11 deg; joints [0.451, -30.232, 97.735, 147.205, 95.577, 27.384, -1.714]
  MoveL 4142 to (-13.55, 61.57, -155.98) mm, rotated rx -167.81 ry 3.47 rz -52.11 deg; joints [0.445, -30.226, 97.704, 147.202, 95.558, 27.399, -1.714]
  MoveL 4143 to (-13.42, 62.02, -155.98) mm, rotated rx -167.81 ry 3.47 rz -52.11 deg; joints [0.44, -30.217, 97.666, 147.198, 95.534, 27.417, -1.714]
  MoveL 4144 to (-13.02, 63.54, -155.98) mm, rotated rx -167.81 ry 3.47 rz -52.11 deg; joints [0.421, -30.188, 97.537, 147.186, 95.455, 27.477, -1.714]
  MoveL 4145 to (-12.86, 64.07, -156) mm, rotated rx -167.81 ry 3.47 rz -52.11 deg; joints [0.413, -30.178, 97.493, 147.182, 95.427, 27.498, -1.714]
  MoveL 4146 to (-12.69, 64.6, -156.05) mm, rotated rx -167.81 ry 3.47 rz -52.11 deg; joints [0.405, -30.171, 97.451, 147.176, 95.4, 27.52, -1.714]
  MoveL 4147 to (-12.49, 65.13, -156.13) mm, rotated rx -167.81 ry 3.47 rz -52.11 deg; joints [0.396, -30.164, 97.409, 147.169, 95.372, 27.542, -1.714]
  MoveL 4148 to (-12.31, 65.66, -156.19) mm, rotated rx -167.81 ry 3.47 rz -52.11 deg; joints [0.387, -30.157, 97.367, 147.163, 95.345, 27.564, -1.714]
  MoveL 4149 to (-12.15, 66.17, -156.22) mm, rotated rx -167.81 ry 3.47 rz -52.11 deg; joints [0.38, -30.148, 97.325, 147.159, 95.319, 27.584, -1.714]
  MoveL 4150 to (-12.01, 66.64, -156.24) mm, rotated rx -167.81 ry 3.47 rz -52.11 deg; joints [0.373, -30.14, 97.286, 147.154, 95.294, 27.603, -1.714]
  MoveL 4151 to (-11.86, 67.08, -156.28) mm, rotated rx -167.81 ry 3.47 rz -52.11 deg; joints [0.366, -30.133, 97.251, 147.15, 95.271, 27.621, -1.714]
  MoveL 4152 to (-11.72, 67.49, -156.32) mm, rotated rx -167.81 ry 3.47 rz -52.11 deg; joints [0.36, -30.127, 97.217, 147.145, 95.25, 27.638, -1.714]
  MoveL 4153 to (-11.58, 67.97, -156.33) mm, rotated rx -167.81 ry 3.47 rz -52.11 deg; joints [0.353, -30.118, 97.177, 147.141, 95.225, 27.658, -1.714]
  MoveL 4154 to (-11.42, 68.53, -156.35) mm, rotated rx -167.81 ry 3.47 rz -52.11 deg; joints [0.346, -30.108, 97.13, 147.136, 95.195, 27.68, -1.714]
  MoveL 4155 to (-11.2, 69.2, -156.41) mm, rotated rx -167.81 ry 3.47 rz -52.11 deg; joints [0.335, -30.097, 97.076, 147.129, 95.161, 27.707, -1.714]
  MoveL 4156 to (-11.02, 69.78, -156.43) mm, rotated rx -167.81 ry 3.47 rz -52.11 deg; joints [0.327, -30.087, 97.027, 147.123, 95.131, 27.731, -1.714]
  MoveL 4157 to (-10.47, 71.81, -156.44) mm, rotated rx -167.81 ry 3.47 rz -52.11 deg; joints [0.302, -30.047, 96.854, 147.108, 95.024, 27.812, -1.714]
  MoveL 4158 to (-9.45, 74.54, -156.77) mm, rotated rx -167.81 ry 3.47 rz -52.11 deg; joints [0.255, -30.007, 96.635, 147.074, 94.884, 27.925, -1.714]
  MoveL 4159 to (-8.78, 75.64, -157.18) mm, rotated rx -167.81 ry 3.47 rz -52.11 deg; joints [0.223, -30.003, 96.558, 147.049, 94.829, 27.976, -1.714]
  MoveL 4160 to (-8, 76.58, -157.76) mm, rotated rx -167.81 ry 3.47 rz -52.11 deg; joints [0.187, -30.01, 96.502, 147.02, 94.785, 28.022, -1.714]
  MoveL 4161 to (-6.14, 77.94, -159.41) mm, rotated rx -167.81 ry 3.47 rz -52.11 deg; joints [0.099, -30.057, 96.457, 146.946, 94.726, 28.102, -1.714]
  MoveL 4162 to (-3.86, 78.62, -161.71) mm, rotated rx -167.81 ry 3.47 rz -52.11 deg; joints [-0.009, -30.148, 96.499, 146.852, 94.709, 28.166, -1.714]
  MoveL 4163 to (-1.84, 78.54, -164.02) mm, rotated rx -167.81 ry 3.47 rz -52.11 deg; joints [-0.106, -30.256, 96.605, 146.766, 94.729, 28.199, -1.714]
  MoveL 4164 to (-1.17, 78.2, -164.93) mm, rotated rx -167.81 ry 3.47 rz -52.11 deg; joints [-0.139, -30.305, 96.674, 146.736, 94.753, 28.199, -1.714]
  MoveL 4165 to (-0.73, 77.65, -165.67) mm, rotated rx -167.81 ry 3.47 rz -52.11 deg; joints [-0.162, -30.352, 96.754, 146.714, 94.785, 28.189, -1.714]
  MoveL 4166 to (-0.6, 77.3, -165.98) mm, rotated rx -167.81 ry 3.47 rz -52.11 deg; joints [-0.169, -30.374, 96.798, 146.707, 94.805, 28.179, -1.714]
  MoveL 4167 to (-0.53, 76.9, -166.24) mm, rotated rx -167.81 ry 3.47 rz -52.11 deg; joints [-0.173, -30.396, 96.845, 146.702, 94.827, 28.167, -1.714]
  MoveL 4168 to (-0.56, 75.94, -166.66) mm, rotated rx -167.81 ry 3.47 rz -52.11 deg; joints [-0.175, -30.437, 96.946, 146.698, 94.878, 28.134, -1.714]
  MoveL 4169 to (-0.81, 74.78, -166.9) mm, rotated rx -167.81 ry 3.47 rz -52.11 deg; joints [-0.166, -30.476, 97.059, 146.702, 94.938, 28.09, -1.714]
  MoveL 4170 to (-1.3, 73.42, -166.99) mm, rotated rx -167.81 ry 3.47 rz -52.11 deg; joints [-0.146, -30.511, 97.182, 146.716, 95.007, 28.035, -1.714]
  MoveL 4171 to (-2.69, 70.03, -166.99) mm, rotated rx -167.81 ry 3.47 rz -52.11 deg; joints [-0.088, -30.589, 97.477, 146.756, 95.176, 27.896, -1.714]
  MoveL 4172 to (-2.88, 69.6, -166.97) mm, rotated rx -167.81 ry 3.47 rz -52.11 deg; joints [-0.08, -30.598, 97.513, 146.762, 95.197, 27.878, -1.714]
  MoveL 4173 to (-3.05, 69.23, -166.94) mm, rotated rx -167.81 ry 3.47 rz -52.11 deg; joints [-0.073, -30.605, 97.545, 146.767, 95.216, 27.863, -1.714]
  MoveL 4174 to (-3.24, 68.8, -166.93) mm, rotated rx -167.81 ry 3.47 rz -52.11 deg; joints [-0.065, -30.614, 97.582, 146.773, 95.237, 27.845, -1.714]
  MoveL 4175 to (-4.64, 65.41, -166.93) mm, rotated rx -167.81 ry 3.47 rz -52.11 deg; joints [-0.006, -30.691, 97.876, 146.814, 95.407, 27.706, -1.714]
  MoveL 4176 to (-4.87, 64.91, -166.9) mm, rotated rx -167.81 ry 3.47 rz -52.11 deg; joints [0.003, -30.701, 97.918, 146.821, 95.431, 27.686, -1.714]
  MoveL 4177 to (-5.12, 64.43, -166.87) mm, rotated rx -167.81 ry 3.47 rz -52.11 deg; joints [0.014, -30.71, 97.958, 146.829, 95.455, 27.665, -1.714]
  MoveL 4178 to (-5.39, 64.02, -166.82) mm, rotated rx -167.81 ry 3.47 rz -52.11 deg; joints [0.025, -30.719, 97.992, 146.838, 95.474, 27.647, -1.714]
  MoveL 4179 to (-5.63, 63.72, -166.76) mm, rotated rx -167.81 ry 3.47 rz -52.11 deg; joints [0.035, -30.724, 98.016, 146.846, 95.488, 27.634, -1.714]
  MoveL 4180 to (-5.77, 63.6, -166.59) mm, rotated rx -167.81 ry 3.47 rz -52.11 deg; joints [0.043, -30.718, 98.019, 146.852, 95.494, 27.626, -1.714]
  MoveL 4181 to (-5.81, 63.61, -166.27) mm, rotated rx -167.81 ry 3.47 rz -52.11 deg; joints [0.048, -30.698, 98.001, 146.856, 95.495, 27.623, -1.714]
  MoveL 4182 to (-5.73, 63.75, -165.76) mm, rotated rx -167.81 ry 3.47 rz -52.11 deg; joints [0.05, -30.662, 97.962, 146.859, 95.491, 27.624, -1.714]
  MoveL 4183 to (-6.56, 63.87, -164.3) mm, rotated rx -167.81 ry 3.47 rz -52.11 deg; joints [0.096, -30.584, 97.884, 146.899, 95.482, 27.61, -1.714]
  MoveL 4184 to (-10.1, 61.49, -164.3) mm, rotated rx -167.81 ry 3.47 rz -52.11 deg; joints [0.229, -30.686, 98.117, 147.011, 95.563, 27.495, -1.714]
  MoveL 4185 to (-11.8, 60.36, -164.25) mm, rotated rx -167.81 ry 3.47 rz -52.11 deg; joints [0.293, -30.732, 98.224, 147.064, 95.602, 27.441, -1.714]
  MoveL 4186 to (-13.45, 59.27, -164.16) mm, rotated rx -167.81 ry 3.47 rz -52.11 deg; joints [0.355, -30.773, 98.326, 147.117, 95.639, 27.387, -1.714]
  MoveL 4187 to (-15.12, 58.15, -164.08) mm, rotated rx -167.81 ry 3.47 rz -52.11 deg; joints [0.419, -30.816, 98.43, 147.171, 95.678, 27.333, -1.714]
  MoveL 4188 to (-16.76, 57.06, -163.98) mm, rotated rx -167.81 ry 3.47 rz -52.11 deg; joints [0.482, -30.856, 98.531, 147.224, 95.716, 27.28, -1.714]
  MoveL 4189 to (-18.52, 55.91, -163.94) mm, rotated rx -167.81 ry 3.47 rz -52.11 deg; joints [0.549, -30.902, 98.639, 147.28, 95.754, 27.225, -1.714]
  MoveL 4190 to (-20.4, 54.78, -163.9) mm, rotated rx -167.81 ry 3.47 rz -52.11 deg; joints [0.62, -30.952, 98.748, 147.34, 95.79, 27.17, -1.714]
  MoveL 4191 to (-22.43, 53.31, -163.73) mm, rotated rx -167.81 ry 3.47 rz -52.11 deg; joints [0.699, -31, 98.879, 147.406, 95.843, 27.1, -1.714]
  MoveL 4192 to (-24.29, 52.06, -163.49) mm, rotated rx -167.81 ry 3.47 rz -52.11 deg; joints [0.772, -31.036, 98.985, 147.468, 95.887, 27.039, -1.714]
  MoveL 4193 to (-26.12, 50.84, -163.35) mm, rotated rx -167.81 ry 3.47 rz -52.11 deg; joints [0.843, -31.079, 99.094, 147.527, 95.929, 26.981, -1.714]
  MoveL 4194 to (-27.89, 49.65, -163.11) mm, rotated rx -167.81 ry 3.47 rz -52.11 deg; joints [0.913, -31.113, 99.195, 147.586, 95.971, 26.923, -1.714]
  MoveL 4195 to (-29.66, 48.46, -162.99) mm, rotated rx -167.81 ry 3.47 rz -52.11 deg; joints [0.981, -31.155, 99.301, 147.644, 96.012, 26.866, -1.714]
  MoveL 4196 to (-31.42, 47.27, -162.87) mm, rotated rx -167.81 ry 3.47 rz -52.11 deg; joints [1.05, -31.197, 99.408, 147.702, 96.053, 26.81, -1.714]
  MoveL 4197 to (-33.19, 46.06, -162.63) mm, rotated rx -167.81 ry 3.47 rz -52.11 deg; joints [1.12, -31.23, 99.508, 147.761, 96.096, 26.752, -1.714]
  MoveL 4198 to (-34.95, 44.86, -162.51) mm, rotated rx -167.81 ry 3.47 rz -52.11 deg; joints [1.189, -31.272, 99.615, 147.819, 96.137, 26.695, -1.714]
  MoveL 4199 to (-36.71, 43.66, -162.4) mm, rotated rx -167.81 ry 3.47 rz -52.11 deg; joints [1.258, -31.313, 99.721, 147.877, 96.179, 26.639, -1.714]
  MoveL 4200 to (-38.47, 42.46, -162.28) mm, rotated rx -167.81 ry 3.47 rz -52.11 deg; joints [1.327, -31.354, 99.827, 147.935, 96.22, 26.583, -1.714]
  MoveL 4201 to (-40.22, 41.23, -162.05) mm, rotated rx -167.81 ry 3.47 rz -52.11 deg; joints [1.397, -31.388, 99.928, 147.994, 96.264, 26.525, -1.714]
  MoveL 4202 to (-41.98, 40.02, -161.94) mm, rotated rx -167.81 ry 3.47 rz -52.11 deg; joints [1.466, -31.429, 100.034, 148.052, 96.305, 26.469, -1.714]
  MoveL 4203 to (-43.43, 38.98, -161.69) mm, rotated rx -167.81 ry 3.47 rz -52.11 deg; joints [1.524, -31.454, 100.117, 148.101, 96.343, 26.419, -1.714]
  MoveL 4204 to (-44.76, 37.99, -161.37) mm, rotated rx -167.81 ry 3.47 rz -52.11 deg; joints [1.58, -31.47, 100.19, 148.147, 96.381, 26.372, -1.714]
  MoveL 4205 to (-46.01, 37.04, -160.95) mm, rotated rx -167.81 ry 3.47 rz -52.11 deg; joints [1.633, -31.479, 100.254, 148.192, 96.418, 26.326, -1.714]
  MoveL 4206 to (-44.29, 37.33, -159.99) mm, rotated rx -167.81 ry 3.47 rz -52.11 deg; joints [1.581, -31.383, 100.166, 148.144, 96.435, 26.338, -1.714]
  MoveL 4207 to (-44.84, 37.01, -159.86) mm, rotated rx -167.81 ry 3.47 rz -52.11 deg; joints [1.603, -31.389, 100.189, 148.163, 96.445, 26.322, -1.714]
  MoveL 4208 to (-45.37, 36.78, -159.78) mm, rotated rx -167.81 ry 3.47 rz -52.11 deg; joints [1.624, -31.396, 100.208, 148.182, 96.45, 26.31, -1.714]
  MoveL 4209 to (-45.91, 36.67, -159.74) mm, rotated rx -167.81 ry 3.47 rz -52.11 deg; joints [1.644, -31.405, 100.219, 148.2, 96.449, 26.302, -1.714]
  MoveL 4210 to (-46.44, 36.61, -159.72) mm, rotated rx -167.81 ry 3.47 rz -52.11 deg; joints [1.664, -31.415, 100.228, 148.217, 96.444, 26.297, -1.714]
  MoveL 4211 to (-50.11, 36.58, -159.72) mm, rotated rx -167.81 ry 3.47 rz -52.11 deg; joints [1.797, -31.482, 100.259, 148.339, 96.388, 26.274, -1.714]
  MoveL 4212 to (-50.58, 36.57, -159.7) mm, rotated rx -167.81 ry 3.47 rz -52.11 deg; joints [1.814, -31.49, 100.263, 148.354, 96.381, 26.271, -1.714]
  MoveL 4213 to (-51, 36.55, -159.68) mm, rotated rx -167.81 ry 3.47 rz -52.11 deg; joints [1.829, -31.496, 100.267, 148.368, 96.376, 26.268, -1.714]
  MoveL 4214 to (-51.48, 36.54, -159.67) mm, rotated rx -167.81 ry 3.47 rz -52.11 deg; joints [1.847, -31.505, 100.271, 148.384, 96.369, 26.265, -1.714]
  MoveL 4215 to (-52.01, 36.54, -159.67) mm, rotated rx -167.81 ry 3.47 rz -52.11 deg; joints [1.866, -31.514, 100.275, 148.402, 96.361, 26.262, -1.714]
  MoveL 4216 to (-53.58, 36.54, -159.67) mm, rotated rx -167.81 ry 3.47 rz -52.11 deg; joints [1.923, -31.543, 100.287, 148.454, 96.336, 26.253, -1.714]
  MoveL 4217 to (-54.2, 36.53, -159.65) mm, rotated rx -167.81 ry 3.47 rz -52.11 deg; joints [1.946, -31.554, 100.292, 148.475, 96.327, 26.249, -1.714]
  MoveL 4218 to (-54.92, 36.5, -159.61) mm, rotated rx -167.81 ry 3.47 rz -52.11 deg; joints [1.972, -31.565, 100.298, 148.498, 96.318, 26.243, -1.714]
  MoveL 4219 to (-55.56, 36.48, -159.59) mm, rotated rx -167.81 ry 3.47 rz -52.11 deg; joints [1.996, -31.575, 100.303, 148.52, 96.308, 26.239, -1.714]
  MoveL 4220 to (-56.61, 36.48, -159.59) mm, rotated rx -167.81 ry 3.47 rz -52.11 deg; joints [2.033, -31.594, 100.311, 148.555, 96.292, 26.233, -1.714]
  MoveL 4221 to (-58.06, 36.55, -159.67) mm, rotated rx -167.81 ry 3.47 rz -52.11 deg; joints [2.084, -31.625, 100.321, 148.602, 96.264, 26.228, -1.714]
  MoveL 4222 to (-59.22, 36.76, -159.92) mm, rotated rx -167.81 ry 3.47 rz -52.11 deg; joints [2.123, -31.66, 100.327, 148.638, 96.232, 26.231, -1.714]
  MoveL 4223 to (-60.11, 37.1, -160.34) mm, rotated rx -167.81 ry 3.47 rz -52.11 deg; joints [2.149, -31.698, 100.328, 148.663, 96.195, 26.242, -1.714]
  MoveL 4224 to (-60.45, 37.33, -160.62) mm, rotated rx -167.81 ry 3.47 rz -52.11 deg; joints [2.157, -31.719, 100.327, 148.672, 96.175, 26.251, -1.714]
  MoveL 4225 to (-60.72, 37.59, -160.93) mm, rotated rx -167.81 ry 3.47 rz -52.11 deg; joints [2.163, -31.741, 100.325, 148.678, 96.154, 26.262, -1.714]
  MoveL 4226 to (-61.05, 38.21, -161.69) mm, rotated rx -167.81 ry 3.47 rz -52.11 deg; joints [2.163, -31.787, 100.317, 148.682, 96.108, 26.29, -1.714]
  MoveL 4227 to (-61.1, 38.97, -162.61) mm, rotated rx -167.81 ry 3.47 rz -52.11 deg; joints [2.152, -31.837, 100.305, 148.675, 96.058, 26.326, -1.714]
  MoveL 4228 to (-60.35, 40.91, -164.96) mm, rotated rx -167.81 ry 3.47 rz -52.11 deg; joints [2.091, -31.947, 100.268, 148.629, 95.943, 26.422, -1.714]
  MoveL 4229 to (-58.82, 42.79, -167.32) mm, rotated rx -167.81 ry 3.47 rz -52.11 deg; joints [2.002, -32.044, 100.229, 148.556, 95.844, 26.521, -1.714]
  MoveL 4230 to (-56.82, 44.02, -169) mm, rotated rx -167.81 ry 3.47 rz -52.11 deg; joints [1.907, -32.098, 100.203, 148.475, 95.795, 26.594, -1.714]
  MoveL 4231 to (-55.65, 44.39, -169.58) mm, rotated rx -167.81 ry 3.47 rz -52.11 deg; joints [1.857, -32.109, 100.195, 148.431, 95.788, 26.62, -1.714]
  MoveL 4232 to (-54.37, 44.59, -170) mm, rotated rx -167.81 ry 3.47 rz -52.11 deg; joints [1.805, -32.109, 100.191, 148.385, 95.794, 26.639, -1.714]
  MoveL 4233 to (-51.45, 44.51, -170.34) mm, rotated rx -167.81 ry 3.47 rz -52.11 deg; joints [1.696, -32.078, 100.192, 148.286, 95.843, 26.657, -1.714]
  MoveL 4234 to (-48.33, 44.11, -170.34) mm, rotated rx -167.81 ry 3.47 rz -52.11 deg; joints [1.585, -32.026, 100.2, 148.183, 95.916, 26.66, -1.714]
  MoveL 4235 to (-47.36, 44.03, -170.39) mm, rotated rx -167.81 ry 3.47 rz -52.11 deg; joints [1.55, -32.012, 100.201, 148.151, 95.935, 26.664, -1.714]
  MoveL 4236 to (-46.84, 43.96, -170.39) mm, rotated rx -167.81 ry 3.47 rz -52.11 deg; joints [1.531, -32.004, 100.202, 148.134, 95.947, 26.664, -1.714]
  MoveL 4237 to (-46.3, 43.89, -170.39) mm, rotated rx -167.81 ry 3.47 rz -52.11 deg; joints [1.512, -31.995, 100.203, 148.116, 95.959, 26.665, -1.714]
  MoveL 4238 to (-45.74, 43.84, -170.41) mm, rotated rx -167.81 ry 3.47 rz -52.11 deg; joints [1.492, -31.987, 100.204, 148.097, 95.971, 26.667, -1.714]
  MoveL 4239 to (-45.09, 43.79, -170.47) mm, rotated rx -167.81 ry 3.47 rz -52.11 deg; joints [1.468, -31.979, 100.206, 148.075, 95.984, 26.669, -1.714]
  MoveL 4240 to (-44.51, 43.73, -170.5) mm, rotated rx -167.81 ry 3.47 rz -52.11 deg; joints [1.447, -31.971, 100.207, 148.056, 95.996, 26.671, -1.714]
  MoveL 4241 to (-43.99, 43.68, -170.52) mm, rotated rx -167.81 ry 3.47 rz -52.11 deg; joints [1.428, -31.963, 100.208, 148.039, 96.007, 26.672, -1.714]
  MoveL 4242 to (-43.51, 43.64, -170.55) mm, rotated rx -167.81 ry 3.47 rz -52.11 deg; joints [1.411, -31.957, 100.209, 148.023, 96.016, 26.674, -1.714]
  MoveL 4243 to (-43.06, 43.62, -170.6) mm, rotated rx -167.81 ry 3.47 rz -52.11 deg; joints [1.394, -31.952, 100.209, 148.007, 96.024, 26.676, -1.714]
  MoveL 4244 to (-42.6, 43.58, -170.63) mm, rotated rx -167.81 ry 3.47 rz -52.11 deg; joints [1.377, -31.946, 100.21, 147.992, 96.033, 26.678, -1.714]
  MoveL 4245 to (-42.1, 43.53, -170.65) mm, rotated rx -167.81 ry 3.47 rz -52.11 deg; joints [1.359, -31.938, 100.211, 147.975, 96.044, 26.679, -1.714]
  MoveL 4246 to (-41.59, 43.48, -170.65) mm, rotated rx -167.81 ry 3.47 rz -52.11 deg; joints [1.341, -31.93, 100.211, 147.958, 96.055, 26.681, -1.714]
  MoveL 4247 to (-41.07, 43.44, -170.66) mm, rotated rx -167.81 ry 3.47 rz -52.11 deg; joints [1.322, -31.921, 100.209, 147.941, 96.065, 26.682, -1.714]
  MoveL 4248 to (-40.58, 43.47, -170.68) mm, rotated rx -167.81 ry 3.47 rz -52.11 deg; joints [1.304, -31.913, 100.204, 147.925, 96.071, 26.687, -1.714]
  MoveL 4249 to (-40.11, 43.55, -170.71) mm, rotated rx -167.81 ry 3.47 rz -52.11 deg; joints [1.287, -31.905, 100.195, 147.909, 96.073, 26.693, -1.714]
  MoveL 4250 to (-39.68, 43.69, -170.75) mm, rotated rx -167.81 ry 3.47 rz -52.11 deg; joints [1.27, -31.898, 100.182, 147.895, 96.072, 26.701, -1.714]
  MoveL 4251 to (-39.26, 43.86, -170.8) mm, rotated rx -167.81 ry 3.47 rz -52.11 deg; joints [1.254, -31.891, 100.168, 147.881, 96.068, 26.71, -1.714]
  MoveL 4252 to (-40.75, 43.54, -171.77) mm, rotated rx -167.81 ry 3.47 rz -52.11 deg; joints [1.298, -31.984, 100.257, 147.92, 96.056, 26.698, -1.714]
  MoveL 4253 to (-39.29, 44.45, -172.14) mm, rotated rx -167.81 ry 3.47 rz -52.11 deg; joints [1.238, -31.969, 100.19, 147.869, 96.025, 26.745, -1.714]
  MoveL 4254 to (-37.72, 45.36, -172.42) mm, rotated rx -167.81 ry 3.47 rz -52.11 deg; joints [1.175, -31.945, 100.118, 147.816, 95.996, 26.791, -1.714]
  MoveL 4255 to (-36.02, 46.3, -172.62) mm, rotated rx -167.81 ry 3.47 rz -52.11 deg; joints [1.108, -31.913, 100.038, 147.759, 95.969, 26.838, -1.714]
  MoveL 4256 to (-34.13, 47.29, -172.85) mm, rotated rx -167.81 ry 3.47 rz -52.11 deg; joints [1.034, -31.879, 99.953, 147.695, 95.94, 26.888, -1.714]
  MoveL 4257 to (-32.23, 48.26, -172.96) mm, rotated rx -167.81 ry 3.47 rz -52.11 deg; joints [0.961, -31.837, 99.863, 147.633, 95.914, 26.937, -1.714]
  MoveL 4258 to (-30.33, 49.23, -173.08) mm, rotated rx -167.81 ry 3.47 rz -52.11 deg; joints [0.888, -31.795, 99.773, 147.57, 95.888, 26.986, -1.714]
  MoveL 4259 to (-28.43, 50.21, -173.31) mm, rotated rx -167.81 ry 3.47 rz -52.11 deg; joints [0.814, -31.761, 99.688, 147.507, 95.861, 27.037, -1.714]
  MoveL 4260 to (-26.52, 51.18, -173.43) mm, rotated rx -167.81 ry 3.47 rz -52.11 deg; joints [0.742, -31.719, 99.599, 147.445, 95.835, 27.086, -1.714]
  MoveL 4261 to (-24.62, 52.14, -173.54) mm, rotated rx -167.81 ry 3.47 rz -52.11 deg; joints [0.669, -31.677, 99.509, 147.382, 95.809, 27.136, -1.714]
  MoveL 4262 to (-22.71, 53.1, -173.78) mm, rotated rx -167.81 ry 3.47 rz -52.11 deg; joints [0.595, -31.643, 99.425, 147.319, 95.782, 27.186, -1.714]
  MoveL 4263 to (-20.81, 54.06, -173.9) mm, rotated rx -167.81 ry 3.47 rz -52.11 deg; joints [0.522, -31.601, 99.335, 147.257, 95.757, 27.236, -1.714]
  MoveL 4264 to (-18.9, 55.01, -174.02) mm, rotated rx -167.81 ry 3.47 rz -52.11 deg; joints [0.45, -31.559, 99.245, 147.194, 95.731, 27.285, -1.714]
  MoveL 4265 to (-17.09, 55.91, -174.21) mm, rotated rx -167.81 ry 3.47 rz -52.11 deg; joints [0.38, -31.524, 99.164, 147.135, 95.707, 27.332, -1.714]
  MoveL 4266 to (-15.45, 56.72, -174.43) mm, rotated rx -167.81 ry 3.47 rz -52.11 deg; joints [0.317, -31.495, 99.093, 147.08, 95.685, 27.376, -1.714]
  MoveL 4267 to (-13.69, 57.59, -174.53) mm, rotated rx -167.81 ry 3.47 rz -52.11 deg; joints [0.25, -31.456, 99.009, 147.024, 95.661, 27.421, -1.714]
  MoveL 4268 to (-11.79, 58.64, -174.53) mm, rotated rx -167.81 ry 3.47 rz -52.11 deg; joints [0.18, -31.405, 98.904, 146.963, 95.631, 27.474, -1.714]
  MoveL 4269 to (-9.35, 59.83, -174.62) mm, rotated rx -167.81 ry 3.47 rz -52.11 deg; joints [0.088, -31.347, 98.786, 146.885, 95.6, 27.536, -1.714]
  MoveL 4270 to (-7.08, 60.81, -174.86) mm, rotated rx -167.81 ry 3.47 rz -52.11 deg; joints [0.002, -31.304, 98.694, 146.811, 95.577, 27.591, -1.714]
  MoveL 4271 to (-5.25, 61.7, -175.04) mm, rotated rx -167.81 ry 3.47 rz -52.11 deg; joints [-0.068, -31.267, 98.611, 146.751, 95.553, 27.639, -1.714]
  MoveL 4272 to (-3.56, 62.49, -175.37) mm, rotated rx -167.81 ry 3.47 rz -52.11 deg; joints [-0.134, -31.244, 98.545, 146.694, 95.531, 27.684, -1.714]
  MoveL 4273 to (-1.72, 63.38, -175.54) mm, rotated rx -167.81 ry 3.47 rz -52.11 deg; joints [-0.204, -31.206, 98.461, 146.634, 95.507, 27.732, -1.714]
  MoveL 4274 to (0.07, 64.21, -175.74) mm, rotated rx -167.81 ry 3.47 rz -52.11 deg; joints [-0.272, -31.172, 98.383, 146.576, 95.485, 27.778, -1.714]
  MoveL 4275 to (1.83, 65, -176.03) mm, rotated rx -167.81 ry 3.47 rz -52.11 deg; joints [-0.34, -31.145, 98.314, 146.518, 95.465, 27.823, -1.714]
  MoveL 4276 to (2.72, 64.83, -176.8) mm, rotated rx -167.81 ry 3.47 rz -52.11 deg; joints [-0.38, -31.178, 98.357, 146.482, 95.482, 27.831, -1.714]
  MoveL 4277 to (2.52, 64.52, -177.18) mm, rotated rx -167.81 ry 3.47 rz -52.11 deg; joints [-0.376, -31.21, 98.405, 146.484, 95.494, 27.821, -1.714]
  MoveL 4278 to (2.5, 64.44, -177.42) mm, rotated rx -167.81 ry 3.47 rz -52.11 deg; joints [-0.378, -31.227, 98.424, 146.482, 95.496, 27.82, -1.714]
  MoveL 4279 to (2.65, 64.59, -177.55) mm, rotated rx -167.81 ry 3.47 rz -52.11 deg; joints [-0.385, -31.23, 98.417, 146.476, 95.489, 27.828, -1.714]
  MoveL 4280 to (2.96, 65.02, -177.59) mm, rotated rx -167.81 ry 3.47 rz -52.11 deg; joints [-0.398, -31.221, 98.381, 146.467, 95.47, 27.847, -1.714]
  MoveL 4281 to (3.33, 65.57, -177.63) mm, rotated rx -167.81 ry 3.47 rz -52.11 deg; joints [-0.413, -31.208, 98.333, 146.455, 95.444, 27.872, -1.714]
  MoveL 4282 to (4.11, 66.94, -177.63) mm, rotated rx -167.81 ry 3.47 rz -52.11 deg; joints [-0.444, -31.173, 98.212, 146.432, 95.379, 27.929, -1.714]
  MoveL 4283 to (4.38, 67.41, -177.64) mm, rotated rx -167.81 ry 3.47 rz -52.11 deg; joints [-0.455, -31.161, 98.171, 146.424, 95.357, 27.949, -1.714]
  MoveL 4284 to (4.66, 67.86, -177.66) mm, rotated rx -167.81 ry 3.47 rz -52.11 deg; joints [-0.466, -31.15, 98.131, 146.415, 95.335, 27.969, -1.714]
  MoveL 4285 to (4.96, 68.32, -177.71) mm, rotated rx -167.81 ry 3.47 rz -52.11 deg; joints [-0.478, -31.14, 98.092, 146.406, 95.314, 27.989, -1.714]
  MoveL 4286 to (5.28, 68.78, -177.79) mm, rotated rx -167.81 ry 3.47 rz -52.11 deg; joints [-0.492, -31.132, 98.055, 146.395, 95.292, 28.01, -1.714]
  MoveL 4287 to (5.59, 69.24, -177.85) mm, rotated rx -167.81 ry 3.47 rz -52.11 deg; joints [-0.504, -31.123, 98.017, 146.386, 95.271, 28.03, -1.714]
  MoveL 4288 to (5.85, 69.66, -177.87) mm, rotated rx -167.81 ry 3.47 rz -52.11 deg; joints [-0.515, -31.113, 97.98, 146.378, 95.251, 28.048, -1.714]
  MoveL 4289 to (6.09, 70.05, -177.89) mm, rotated rx -167.81 ry 3.47 rz -52.11 deg; joints [-0.524, -31.103, 97.946, 146.37, 95.232, 28.065, -1.714]
  MoveL 4290 to (6.87, 71.42, -177.89) mm, rotated rx -167.81 ry 3.47 rz -52.11 deg; joints [-0.555, -31.068, 97.824, 146.347, 95.167, 28.123, -1.714]
  MoveL 4291 to (7.13, 71.87, -177.9) mm, rotated rx -167.81 ry 3.47 rz -52.11 deg; joints [-0.566, -31.057, 97.785, 146.339, 95.146, 28.142, -1.714]
  MoveL 4292 to (7.39, 72.27, -177.93) mm, rotated rx -167.81 ry 3.47 rz -52.11 deg; joints [-0.576, -31.047, 97.75, 146.332, 95.127, 28.16, -1.714]
  MoveL 4293 to (7.64, 72.63, -177.98) mm, rotated rx -167.81 ry 3.47 rz -52.11 deg; joints [-0.586, -31.04, 97.72, 146.324, 95.11, 28.176, -1.714]
  MoveL 4294 to (7.89, 73.01, -178.01) mm, rotated rx -167.81 ry 3.47 rz -52.11 deg; joints [-0.596, -31.032, 97.687, 146.316, 95.092, 28.193, -1.714]
  MoveL 4295 to (8.14, 73.43, -178.03) mm, rotated rx -167.81 ry 3.47 rz -52.11 deg; joints [-0.606, -31.021, 97.65, 146.308, 95.073, 28.211, -1.714]
  MoveL 4296 to (8.4, 73.89, -178.03) mm, rotated rx -167.81 ry 3.47 rz -52.11 deg; joints [-0.617, -31.009, 97.61, 146.3, 95.051, 28.23, -1.714]
  MoveL 4297 to (10.1, 76.27, -178.37) mm, rotated rx -167.81 ry 3.47 rz -52.11 deg; joints [-0.686, -30.96, 97.409, 146.246, 94.94, 28.338, -1.714]
  MoveL 4298 to (11.05, 77.19, -178.79) mm, rotated rx -167.81 ry 3.47 rz -52.11 deg; joints [-0.726, -30.954, 97.344, 146.213, 94.9, 28.384, -1.714]
  MoveL 4299 to (12.06, 77.92, -179.38) mm, rotated rx -167.81 ry 3.47 rz -52.11 deg; joints [-0.77, -30.96, 97.302, 146.176, 94.87, 28.426, -1.714]
  MoveL 4300 to (14.27, 78.82, -181.07) mm, rotated rx -167.81 ry 3.47 rz -52.11 deg; joints [-0.87, -31.009, 97.288, 146.091, 94.841, 28.494, -1.714]
  MoveL 4301 to (16.73, 78.98, -183.43) mm, rotated rx -167.81 ry 3.47 rz -52.11 deg; joints [-0.984, -31.106, 97.367, 145.991, 94.851, 28.543, -1.714]
  MoveL 4302 to (18.75, 78.48, -185.79) mm, rotated rx -167.81 ry 3.47 rz -52.11 deg; joints [-1.082, -31.221, 97.505, 145.903, 94.892, 28.563, -1.714]
  MoveL 4303 to (19.34, 78.01, -186.72) mm, rotated rx -167.81 ry 3.47 rz -52.11 deg; joints [-1.113, -31.275, 97.585, 145.874, 94.92, 28.559, -1.714]
  MoveL 4304 to (19.65, 77.39, -187.48) mm, rotated rx -167.81 ry 3.47 rz -52.11 deg; joints [-1.131, -31.326, 97.671, 145.856, 94.953, 28.545, -1.714]
  MoveL 4305 to (19.7, 77.03, -187.8) mm, rotated rx -167.81 ry 3.47 rz -52.11 deg; joints [-1.136, -31.351, 97.716, 145.851, 94.972, 28.535, -1.714]
  MoveL 4306 to (19.68, 76.64, -188.07) mm, rotated rx -167.81 ry 3.47 rz -52.11 deg; joints [-1.138, -31.374, 97.764, 145.848, 94.992, 28.522, -1.714]
  MoveL 4307 to (19.42, 75.73, -188.49) mm, rotated rx -167.81 ry 3.47 rz -52.11 deg; joints [-1.132, -31.42, 97.863, 145.851, 95.035, 28.489, -1.714]
  MoveL 4308 to (18.89, 74.68, -188.74) mm, rotated rx -167.81 ry 3.47 rz -52.11 deg; joints [-1.114, -31.463, 97.97, 145.864, 95.084, 28.448, -1.714]
  MoveL 4309 to (18.07, 73.49, -188.83) mm, rotated rx -167.81 ry 3.47 rz -52.11 deg; joints [-1.084, -31.502, 98.083, 145.887, 95.138, 28.396, -1.714]
  MoveL 4310 to (17.12, 72.24, -188.83) mm, rotated rx -167.81 ry 3.47 rz -52.11 deg; joints [-1.047, -31.54, 98.198, 145.915, 95.194, 28.341, -1.714]
  MoveL 4311 to (16.8, 71.82, -188.82) mm, rotated rx -167.81 ry 3.47 rz -52.11 deg; joints [-1.035, -31.553, 98.236, 145.924, 95.213, 28.322, -1.714]
  MoveL 4312 to (16.43, 71.37, -188.79) mm, rotated rx -167.81 ry 3.47 rz -52.11 deg; joints [-1.021, -31.565, 98.276, 145.936, 95.232, 28.302, -1.714]
  MoveL 4313 to (16.01, 70.89, -188.72) mm, rotated rx -167.81 ry 3.47 rz -52.11 deg; joints [-1.004, -31.576, 98.317, 145.949, 95.253, 28.28, -1.714]
  MoveL 4314 to (15.65, 70.45, -188.7) mm, rotated rx -167.81 ry 3.47 rz -52.11 deg; joints [-0.99, -31.588, 98.357, 145.96, 95.273, 28.26, -1.714]
  MoveL 4315 to (15.33, 70.03, -188.7) mm, rotated rx -167.81 ry 3.47 rz -52.11 deg; joints [-0.978, -31.601, 98.395, 145.97, 95.292, 28.241, -1.714]
  MoveL 4316 to (15.01, 69.62, -188.69) mm, rotated rx -167.81 ry 3.47 rz -52.11 deg; joints [-0.966, -31.613, 98.432, 145.979, 95.31, 28.223, -1.714]
  MoveL 4317 to (14.68, 69.23, -188.64) mm, rotated rx -167.81 ry 3.47 rz -52.11 deg; joints [-0.952, -31.622, 98.466, 145.99, 95.327, 28.205, -1.714]
  MoveL 4318 to (14.34, 68.87, -188.56) mm, rotated rx -167.81 ry 3.47 rz -52.11 deg; joints [-0.939, -31.629, 98.496, 146.001, 95.343, 28.188, -1.714]
  MoveL 4319 to (13.98, 68.51, -188.47) mm, rotated rx -167.81 ry 3.47 rz -52.11 deg; joints [-0.924, -31.636, 98.525, 146.013, 95.358, 28.17, -1.714]
  MoveL 4320 to (13.64, 68.13, -188.4) mm, rotated rx -167.81 ry 3.47 rz -52.11 deg; joints [-0.91, -31.644, 98.557, 146.024, 95.375, 28.152, -1.714]
  MoveL 4321 to (13.3, 67.72, -188.36) mm, rotated rx -167.81 ry 3.47 rz -52.11 deg; joints [-0.897, -31.655, 98.593, 146.034, 95.393, 28.134, -1.714]
  MoveL 4322 to (12.98, 67.31, -188.35) mm, rotated rx -167.81 ry 3.47 rz -52.11 deg; joints [-0.885, -31.666, 98.63, 146.044, 95.411, 28.116, -1.714]
  MoveL 4323 to (11.4, 65.29, -188.35) mm, rotated rx -167.81 ry 3.47 rz -52.11 deg; joints [-0.824, -31.727, 98.814, 146.091, 95.501, 28.027, -1.714]
  MoveL 4324 to (11.13, 65.03, -188.32) mm, rotated rx -167.81 ry 3.47 rz -52.11 deg; joints [-0.813, -31.735, 98.838, 146.1, 95.512, 28.014, -1.714]
  MoveL 4325 to (10.99, 64.93, -188.21) mm, rotated rx -167.81 ry 3.47 rz -52.11 deg; joints [-0.807, -31.732, 98.841, 146.105, 95.516, 28.008, -1.714]
  MoveL 4326 to (11.05, 64.99, -187.98) mm, rotated rx -167.81 ry 3.47 rz -52.11 deg; joints [-0.807, -31.715, 98.824, 146.105, 95.515, 28.009, -1.714]
  MoveL 4327 to (11.33, 65.22, -187.61) mm, rotated rx -167.81 ry 3.47 rz -52.11 deg; joints [-0.813, -31.683, 98.784, 146.1, 95.509, 28.016, -1.714]
  MoveL 4328 to (10.59, 65.4, -186.88) mm, rotated rx -167.81 ry 3.47 rz -52.11 deg; joints [-0.778, -31.649, 98.739, 146.132, 95.494, 28.01, -1.714]
  MoveL 4329 to (8.58, 64.71, -186.86) mm, rotated rx -167.81 ry 3.47 rz -52.11 deg; joints [-0.705, -31.698, 98.818, 146.195, 95.503, 27.969, -1.714]
  MoveL 4330 to (6.51, 64.03, -186.73) mm, rotated rx -167.81 ry 3.47 rz -52.11 deg; joints [-0.628, -31.74, 98.892, 146.262, 95.512, 27.927, -1.714]
  MoveL 4331 to (4.33, 63.36, -186.47) mm, rotated rx -167.81 ry 3.47 rz -52.11 deg; joints [-0.546, -31.776, 98.958, 146.334, 95.52, 27.883, -1.714]
  MoveL 4332 to (2.32, 62.7, -186.33) mm, rotated rx -167.81 ry 3.47 rz -52.11 deg; joints [-0.471, -31.817, 99.028, 146.399, 95.528, 27.843, -1.714]
  MoveL 4333 to (0.38, 62.07, -186.07) mm, rotated rx -167.81 ry 3.47 rz -52.11 deg; joints [-0.397, -31.847, 99.088, 146.463, 95.537, 27.802, -1.714]
  MoveL 4334 to (-1.63, 61.43, -185.72) mm, rotated rx -167.81 ry 3.47 rz -52.11 deg; joints [-0.32, -31.873, 99.144, 146.53, 95.545, 27.761, -1.714]
  MoveL 4335 to (-3.67, 60.75, -185.58) mm, rotated rx -167.81 ry 3.47 rz -52.11 deg; joints [-0.244, -31.914, 99.215, 146.597, 95.554, 27.719, -1.714]
  MoveL 4336 to (-5.67, 60.07, -185.48) mm, rotated rx -167.81 ry 3.47 rz -52.11 deg; joints [-0.169, -31.956, 99.287, 146.661, 95.563, 27.679, -1.714]
  MoveL 4337 to (-7.7, 59.38, -185.33) mm, rotated rx -167.81 ry 3.47 rz -52.11 deg; joints [-0.093, -31.996, 99.358, 146.728, 95.573, 27.637, -1.714]
  MoveL 4338 to (-9.69, 58.73, -185.04) mm, rotated rx -167.81 ry 3.47 rz -52.11 deg; joints [-0.017, -32.026, 99.416, 146.794, 95.581, 27.596, -1.714]
  MoveL 4339 to (-11.74, 57.98, -184.71) mm, rotated rx -167.81 ry 3.47 rz -52.11 deg; joints [0.063, -32.054, 99.481, 146.863, 95.595, 27.551, -1.714]
  MoveL 4340 to (-13.75, 57.28, -184.52) mm, rotated rx -167.81 ry 3.47 rz -52.11 deg; joints [0.138, -32.091, 99.55, 146.929, 95.605, 27.509, -1.714]
  MoveL 4341 to (-15.77, 56.57, -184.42) mm, rotated rx -167.81 ry 3.47 rz -52.11 deg; joints [0.214, -32.133, 99.622, 146.995, 95.615, 27.468, -1.714]
  MoveL 4342 to (-17.78, 55.87, -184.34) mm, rotated rx -167.81 ry 3.47 rz -52.11 deg; joints [0.289, -32.177, 99.696, 147.06, 95.624, 27.428, -1.714]
  MoveL 4343 to (-19.79, 55.15, -184.12) mm, rotated rx -167.81 ry 3.47 rz -52.11 deg; joints [0.366, -32.212, 99.763, 147.127, 95.636, 27.385, -1.714]
  MoveL 4344 to (-21.79, 54.44, -183.98) mm, rotated rx -167.81 ry 3.47 rz -52.11 deg; joints [0.441, -32.251, 99.834, 147.192, 95.646, 27.344, -1.714]
  MoveL 4345 to (-23.81, 53.72, -183.91) mm, rotated rx -167.81 ry 3.47 rz -52.11 deg; joints [0.517, -32.295, 99.907, 147.258, 95.656, 27.303, -1.714]
  MoveL 4346 to (-25.81, 52.99, -183.68) mm, rotated rx -167.81 ry 3.47 rz -52.11 deg; joints [0.593, -32.329, 99.974, 147.325, 95.668, 27.261, -1.714]
  MoveL 4347 to (-27.82, 52.23, -183.44) mm, rotated rx -167.81 ry 3.47 rz -52.11 deg; joints [0.671, -32.362, 100.042, 147.392, 95.681, 27.217, -1.714]
  MoveL 4348 to (-29.87, 51.49, -183.29) mm, rotated rx -167.81 ry 3.47 rz -52.11 deg; joints [0.748, -32.402, 100.114, 147.46, 95.692, 27.175, -1.714]
  MoveL 4349 to (-31.62, 50.81, -183.17) mm, rotated rx -167.81 ry 3.47 rz -52.11 deg; joints [0.815, -32.437, 100.178, 147.518, 95.704, 27.137, -1.714]
  MoveL 4350 to (-33.13, 50.17, -182.96) mm, rotated rx -167.81 ry 3.47 rz -52.11 deg; joints [0.874, -32.46, 100.233, 147.569, 95.718, 27.102, -1.714]
  MoveL 4351 to (-34.42, 49.54, -182.64) mm, rotated rx -167.81 ry 3.47 rz -52.11 deg; joints [0.926, -32.473, 100.279, 147.613, 95.736, 27.067, -1.714]
  MoveL 4352 to (-32.97, 49.8, -181.68) mm, rotated rx -167.81 ry 3.47 rz -52.11 deg; joints [0.884, -32.382, 100.196, 147.575, 95.751, 27.076, -1.714]
  MoveL 4353 to (-33.44, 49.64, -181.68) mm, rotated rx -167.81 ry 3.47 rz -52.11 deg; joints [0.901, -32.393, 100.213, 147.591, 95.753, 27.067, -1.714]
  MoveL 4354 to (-33.92, 49.52, -181.67) mm, rotated rx -167.81 ry 3.47 rz -52.11 deg; joints [0.919, -32.403, 100.227, 147.606, 95.752, 27.059, -1.714]
  MoveL 4355 to (-34.45, 49.48, -181.65) mm, rotated rx -167.81 ry 3.47 rz -52.11 deg; joints [0.939, -32.412, 100.234, 147.624, 95.746, 27.055, -1.714]
  MoveL 4356 to (-35.02, 49.5, -181.61) mm, rotated rx -167.81 ry 3.47 rz -52.11 deg; joints [0.959, -32.42, 100.234, 147.643, 95.736, 27.052, -1.714]
  MoveL 4357 to (-35.62, 49.58, -181.55) mm, rotated rx -167.81 ry 3.47 rz -52.11 deg; joints [0.981, -32.426, 100.231, 147.663, 95.723, 27.05, -1.714]
  MoveL 4358 to (-36.19, 49.7, -181.51) mm, rotated rx -167.81 ry 3.47 rz -52.11 deg; joints [1.002, -32.433, 100.224, 147.682, 95.708, 27.05, -1.714]
  MoveL 4359 to (-36.74, 49.83, -181.5) mm, rotated rx -167.81 ry 3.47 rz -52.11 deg; joints [1.021, -32.44, 100.218, 147.7, 95.692, 27.052, -1.714]
  MoveL 4360 to (-37.25, 49.96, -181.5) mm, rotated rx -167.81 ry 3.47 rz -52.11 deg; joints [1.039, -32.448, 100.211, 147.717, 95.677, 27.054, -1.714]
  MoveL 4361 to (-37.76, 50.09, -181.49) mm, rotated rx -167.81 ry 3.47 rz -52.11 deg; joints [1.057, -32.455, 100.205, 147.734, 95.661, 27.055, -1.714]
  MoveL 4362 to (-38.33, 50.21, -181.45) mm, rotated rx -167.81 ry 3.47 rz -52.11 deg; joints [1.078, -32.462, 100.198, 147.753, 95.646, 27.056, -1.714]
  MoveL 4363 to (-38.98, 50.32, -181.36) mm, rotated rx -167.81 ry 3.47 rz -52.11 deg; joints [1.102, -32.467, 100.191, 147.775, 95.63, 27.055, -1.714]
  MoveL 4364 to (-39.49, 50.42, -181.32) mm, rotated rx -167.81 ry 3.47 rz -52.11 deg; joints [1.121, -32.472, 100.184, 147.792, 95.617, 27.055, -1.714]
  MoveL 4365 to (-39.91, 50.51, -181.29) mm, rotated rx -167.81 ry 3.47 rz -52.11 deg; joints [1.135, -32.477, 100.179, 147.806, 95.606, 27.055, -1.714]
  MoveL 4366 to (-40.37, 50.63, -181.28) mm, rotated rx -167.81 ry 3.47 rz -52.11 deg; joints [1.152, -32.483, 100.173, 147.822, 95.592, 27.057, -1.714]
  MoveL 4367 to (-40.88, 50.76, -181.27) mm, rotated rx -167.81 ry 3.47 rz -52.11 deg; joints [1.17, -32.49, 100.166, 147.838, 95.576, 27.058, -1.714]
  MoveL 4368 to (-41.37, 50.88, -181.26) mm, rotated rx -167.81 ry 3.47 rz -52.11 deg; joints [1.187, -32.497, 100.16, 147.854, 95.562, 27.059, -1.714]
  MoveL 4369 to (-41.86, 50.99, -181.23) mm, rotated rx -167.81 ry 3.47 rz -52.11 deg; joints [1.205, -32.503, 100.154, 147.871, 95.548, 27.06, -1.714]
  MoveL 4370 to (-42.35, 51.11, -181.22) mm, rotated rx -167.81 ry 3.47 rz -52.11 deg; joints [1.222, -32.51, 100.148, 147.887, 95.534, 27.061, -1.714]
  MoveL 4371 to (-44.9, 51.78, -181.22) mm, rotated rx -167.81 ry 3.47 rz -52.11 deg; joints [1.312, -32.547, 100.114, 147.97, 95.456, 27.07, -1.714]
  MoveL 4372 to (-46.28, 52.21, -181.3) mm, rotated rx -167.81 ry 3.47 rz -52.11 deg; joints [1.359, -32.572, 100.095, 148.015, 95.409, 27.078, -1.714]
  MoveL 4373 to (-47.38, 52.7, -181.55) mm, rotated rx -167.81 ry 3.47 rz -52.11 deg; joints [1.394, -32.601, 100.077, 148.048, 95.362, 27.092, -1.714]
  MoveL 4374 to (-48.18, 53.25, -181.97) mm, rotated rx -167.81 ry 3.47 rz -52.11 deg; joints [1.416, -32.634, 100.06, 148.071, 95.315, 27.111, -1.714]
  MoveL 4375 to (-48.68, 53.85, -182.55) mm, rotated rx -167.81 ry 3.47 rz -52.11 deg; joints [1.425, -32.672, 100.045, 148.082, 95.268, 27.136, -1.714]
  MoveL 4376 to (-48.89, 54.51, -183.3) mm, rotated rx -167.81 ry 3.47 rz -52.11 deg; joints [1.422, -32.714, 100.032, 148.082, 95.222, 27.167, -1.714]
  MoveL 4377 to (-48.81, 55.23, -184.22) mm, rotated rx -167.81 ry 3.47 rz -52.11 deg; joints [1.406, -32.76, 100.019, 148.07, 95.175, 27.203, -1.714]
  MoveL 4378 to (-47.76, 56.84, -186.55) mm, rotated rx -167.81 ry 3.47 rz -52.11 deg; joints [1.337, -32.865, 99.999, 148.014, 95.083, 27.292, -1.714]
  MoveL 4379 to (-45.95, 58.22, -188.89) mm, rotated rx -167.81 ry 3.47 rz -52.11 deg; joints [1.241, -32.959, 99.991, 147.933, 95.016, 27.379, -1.714]
  MoveL 4380 to (-43.8, 58.93, -190.6) mm, rotated rx -167.81 ry 3.47 rz -52.11 deg; joints [1.142, -33.017, 100.002, 147.847, 94.997, 27.437, -1.714]
  MoveL 4381 to (-42.59, 59.03, -191.22) mm, rotated rx -167.81 ry 3.47 rz -52.11 deg; joints [1.091, -33.032, 100.015, 147.802, 95.006, 27.455, -1.714]
  MoveL 4382 to (-41.3, 58.96, -191.67) mm, rotated rx -167.81 ry 3.47 rz -52.11 deg; joints [1.04, -33.037, 100.032, 147.756, 95.027, 27.465, -1.714]
  MoveL 4383 to (-38.45, 58.32, -192.1) mm, rotated rx -167.81 ry 3.47 rz -52.11 deg; joints [0.935, -33.021, 100.082, 147.659, 95.104, 27.465, -1.714]
  MoveL 4384 to (-37.49, 58.01, -192.14) mm, rotated rx -167.81 ry 3.47 rz -52.11 deg; joints [0.901, -33.01, 100.101, 147.627, 95.137, 27.46, -1.714]
  MoveL 4385 to (-35.06, 57.03, -192.14) mm, rotated rx -167.81 ry 3.47 rz -52.11 deg; joints [0.817, -32.979, 100.16, 147.548, 95.23, 27.439, -1.714]
  MoveL 4386 to (-34.12, 56.69, -192.19) mm, rotated rx -167.81 ry 3.47 rz -52.11 deg; joints [0.783, -32.97, 100.182, 147.517, 95.264, 27.433, -1.714]
  MoveL 4387 to (-33.14, 56.29, -192.19) mm, rotated rx -167.81 ry 3.47 rz -52.11 deg; joints [0.749, -32.957, 100.205, 147.485, 95.301, 27.425, -1.714]
  MoveL 4388 to (-32.69, 56.12, -192.2) mm, rotated rx -167.81 ry 3.47 rz -52.11 deg; joints [0.734, -32.952, 100.216, 147.47, 95.318, 27.421, -1.714]
  MoveL 4389 to (-32.29, 55.98, -192.23) mm, rotated rx -167.81 ry 3.47 rz -52.11 deg; joints [0.719, -32.948, 100.225, 147.456, 95.332, 27.419, -1.714]
  MoveL 4390 to (-31.85, 55.81, -192.24) mm, rotated rx -167.81 ry 3.47 rz -52.11 deg; joints [0.704, -32.943, 100.236, 147.442, 95.348, 27.416, -1.714]
  MoveL 4391 to (-29.43, 54.83, -192.25) mm, rotated rx -167.81 ry 3.47 rz -52.11 deg; joints [0.62, -32.912, 100.293, 147.362, 95.441, 27.395, -1.714]
  MoveL 4392 to (-28.96, 54.66, -192.26) mm, rotated rx -167.81 ry 3.47 rz -52.11 deg; joints [0.603, -32.906, 100.304, 147.347, 95.457, 27.392, -1.714]
  MoveL 4393 to (-28.52, 54.52, -192.3) mm, rotated rx -167.81 ry 3.47 rz -52.11 deg; joints [0.587, -32.902, 100.313, 147.332, 95.472, 27.39, -1.714]
  MoveL 4394 to (-28.09, 54.42, -192.34) mm, rotated rx -167.81 ry 3.47 rz -52.11 deg; joints [0.572, -32.898, 100.319, 147.318, 95.483, 27.389, -1.714]
  MoveL 4395 to (-27.66, 54.36, -192.38) mm, rotated rx -167.81 ry 3.47 rz -52.11 deg; joints [0.556, -32.893, 100.322, 147.303, 95.493, 27.39, -1.714]
  MoveL 4396 to (-27.22, 54.36, -192.39) mm, rotated rx -167.81 ry 3.47 rz -52.11 deg; joints [0.54, -32.886, 100.318, 147.289, 95.5, 27.393, -1.714]
  MoveL 4397 to (-26.78, 54.41, -192.4) mm, rotated rx -167.81 ry 3.47 rz -52.11 deg; joints [0.524, -32.877, 100.311, 147.274, 95.504, 27.398, -1.714]
  MoveL 4398 to (-27.54, 54.46, -193.13) mm, rotated rx -167.81 ry 3.47 rz -52.11 deg; joints [0.543, -32.937, 100.351, 147.292, 95.483, 27.403, -1.714]
  MoveL 4399 to (-26.21, 55, -193.69) mm, rotated rx -167.81 ry 3.47 rz -52.11 deg; joints [0.487, -32.939, 100.323, 147.244, 95.47, 27.437, -1.714]
  MoveL 4400 to (-24.73, 55.49, -194.11) mm, rotated rx -167.81 ry 3.47 rz -52.11 deg; joints [0.427, -32.931, 100.29, 147.192, 95.462, 27.47, -1.714]
  MoveL 4401 to (-23.02, 55.96, -194.42) mm, rotated rx -167.81 ry 3.47 rz -52.11 deg; joints [0.361, -32.911, 100.251, 147.134, 95.459, 27.502, -1.714]
  MoveL 4402 to (-21.06, 56.42, -194.6) mm, rotated rx -167.81 ry 3.47 rz -52.11 deg; joints [0.287, -32.879, 100.204, 147.068, 95.463, 27.534, -1.714]
  MoveL 4403 to (-19.01, 56.89, -194.8) mm, rotated rx -167.81 ry 3.47 rz -52.11 deg; joints [0.21, -32.845, 100.156, 147, 95.466, 27.567, -1.714]
  MoveL 4404 to (-16.93, 57.34, -194.91) mm, rotated rx -167.81 ry 3.47 rz -52.11 deg; joints [0.132, -32.806, 100.104, 146.932, 95.472, 27.599, -1.714]
  MoveL 4405 to (-14.84, 57.8, -195.14) mm, rotated rx -167.81 ry 3.47 rz -52.11 deg; joints [0.054, -32.774, 100.057, 146.863, 95.476, 27.633, -1.714]
  MoveL 4406 to (-12.76, 58.25, -195.26) mm, rotated rx -167.81 ry 3.47 rz -52.11 deg; joints [-0.024, -32.735, 100.005, 146.794, 95.482, 27.665, -1.714]
  MoveL 4407 to (-10.67, 58.7, -195.37) mm, rotated rx -167.81 ry 3.47 rz -52.11 deg; joints [-0.101, -32.695, 99.954, 146.726, 95.488, 27.697, -1.714]
  MoveL 4408 to (-8.58, 59.14, -195.49) mm, rotated rx -167.81 ry 3.47 rz -52.11 deg; joints [-0.178, -32.656, 99.902, 146.658, 95.494, 27.729, -1.714]
  MoveL 4409 to (-6.49, 59.58, -195.73) mm, rotated rx -167.81 ry 3.47 rz -52.11 deg; joints [-0.257, -32.624, 99.855, 146.588, 95.499, 27.762, -1.714]
  MoveL 4410 to (-4.41, 60.02, -195.84) mm, rotated rx -167.81 ry 3.47 rz -52.11 deg; joints [-0.335, -32.584, 99.803, 146.52, 95.505, 27.794, -1.714]
  MoveL 4411 to (-2.41, 60.5, -195.95) mm, rotated rx -167.81 ry 3.47 rz -52.11 deg; joints [-0.408, -32.545, 99.748, 146.455, 95.507, 27.827, -1.714]
  MoveL 4412 to (-0.48, 61.08, -196.15) mm, rotated rx -167.81 ry 3.47 rz -52.11 deg; joints [-0.481, -32.512, 99.69, 146.391, 95.502, 27.865, -1.714]
  MoveL 4413 to (1.97, 61.56, -196.29) mm, rotated rx -167.81 ry 3.47 rz -52.11 deg; joints [-0.572, -32.466, 99.63, 146.311, 95.51, 27.902, -1.714]
  MoveL 4414 to (4.4, 61.91, -196.38) mm, rotated rx -167.81 ry 3.47 rz -52.11 deg; joints [-0.66, -32.419, 99.579, 146.233, 95.526, 27.933, -1.714]
  MoveL 4415 to (6.65, 62.3, -196.41) mm, rotated rx -167.81 ry 3.47 rz -52.11 deg; joints [-0.742, -32.371, 99.523, 146.16, 95.537, 27.964, -1.714]
  MoveL 4416 to (8.67, 62.7, -196.45) mm, rotated rx -167.81 ry 3.47 rz -52.11 deg; joints [-0.816, -32.328, 99.469, 146.096, 95.544, 27.994, -1.714]
  MoveL 4417 to (10.59, 63.1, -196.57) mm, rotated rx -167.81 ry 3.47 rz -52.11 deg; joints [-0.887, -32.292, 99.42, 146.033, 95.549, 28.024, -1.714]
  MoveL 4418 to (12.57, 63.51, -196.64) mm, rotated rx -167.81 ry 3.47 rz -52.11 deg; joints [-0.959, -32.251, 99.367, 145.969, 95.554, 28.054, -1.714]
  MoveL 4419 to (14.66, 63.93, -196.71) mm, rotated rx -167.81 ry 3.47 rz -52.11 deg; joints [-1.035, -32.208, 99.311, 145.902, 95.56, 28.086, -1.714]
  MoveL 4420 to (16.61, 64.3, -196.89) mm, rotated rx -167.81 ry 3.47 rz -52.11 deg; joints [-1.108, -32.175, 99.266, 145.838, 95.566, 28.116, -1.714]
  MoveL 4421 to (18.48, 64.63, -197.21) mm, rotated rx -167.81 ry 3.47 rz -52.11 deg; joints [-1.179, -32.152, 99.232, 145.775, 95.572, 28.146, -1.714]
  MoveL 4422 to (19.3, 64.34, -198.25) mm, rotated rx -167.81 ry 3.47 rz -52.11 deg; joints [-1.22, -32.206, 99.299, 145.738, 95.592, 28.152, -1.714]
  MoveL 4423 to (19.07, 64.23, -198.76) mm, rotated rx -167.81 ry 3.47 rz -52.11 deg; joints [-1.218, -32.244, 99.336, 145.741, 95.591, 28.151, -1.714]
  MoveL 4424 to (19.06, 64.21, -199.09) mm, rotated rx -167.81 ry 3.47 rz -52.11 deg; joints [-1.221, -32.265, 99.354, 145.738, 95.589, 28.154, -1.714]
  MoveL 4425 to (19.27, 64.27, -199.25) mm, rotated rx -167.81 ry 3.47 rz -52.11 deg; joints [-1.231, -32.27, 99.355, 145.73, 95.588, 28.159, -1.714]
  MoveL 4426 to (19.65, 64.45, -199.29) mm, rotated rx -167.81 ry 3.47 rz -52.11 deg; joints [-1.245, -32.262, 99.337, 145.717, 95.583, 28.17, -1.714]
  MoveL 4427 to (20.09, 64.73, -199.3) mm, rotated rx -167.81 ry 3.47 rz -52.11 deg; joints [-1.261, -32.25, 99.31, 145.703, 95.574, 28.184, -1.714]
  MoveL 4428 to (20.55, 65.11, -199.31) mm, rotated rx -167.81 ry 3.47 rz -52.11 deg; joints [-1.279, -32.236, 99.274, 145.689, 95.559, 28.202, -1.714]
  MoveL 4429 to (21.01, 65.53, -199.33) mm, rotated rx -167.81 ry 3.47 rz -52.11 deg; joints [-1.296, -32.221, 99.234, 145.675, 95.542, 28.222, -1.714]
  MoveL 4430 to (23.58, 68.15, -199.33) mm, rotated rx -167.81 ry 3.47 rz -52.11 deg; joints [-1.392, -32.131, 98.987, 145.598, 95.434, 28.342, -1.714]
  MoveL 4431 to (23.9, 68.45, -199.35) mm, rotated rx -167.81 ry 3.47 rz -52.11 deg; joints [-1.405, -32.122, 98.959, 145.588, 95.422, 28.356, -1.714]
  MoveL 4432 to (24.24, 68.8, -199.36) mm, rotated rx -167.81 ry 3.47 rz -52.11 deg; joints [-1.418, -32.11, 98.927, 145.578, 95.408, 28.372, -1.714]
  MoveL 4433 to (24.61, 69.17, -199.37) mm, rotated rx -167.81 ry 3.47 rz -52.11 deg; joints [-1.431, -32.098, 98.892, 145.567, 95.392, 28.389, -1.714]
  MoveL 4434 to (24.96, 69.51, -199.39) mm, rotated rx -167.81 ry 3.47 rz -52.11 deg; joints [-1.445, -32.087, 98.861, 145.556, 95.379, 28.405, -1.714]
  MoveL 4435 to (25.31, 69.82, -199.43) mm, rotated rx -167.81 ry 3.47 rz -52.11 deg; joints [-1.458, -32.077, 98.833, 145.545, 95.366, 28.42, -1.714]
  MoveL 4436 to (25.63, 70.1, -199.48) mm, rotated rx -167.81 ry 3.47 rz -52.11 deg; joints [-1.471, -32.07, 98.809, 145.535, 95.355, 28.434, -1.714]
  MoveL 4437 to (25.98, 70.42, -199.52) mm, rotated rx -167.81 ry 3.47 rz -52.11 deg; joints [-1.484, -32.061, 98.78, 145.524, 95.342, 28.45, -1.714]
  MoveL 4438 to (26.33, 70.75, -199.54) mm, rotated rx -167.81 ry 3.47 rz -52.11 deg; joints [-1.497, -32.05, 98.748, 145.513, 95.328, 28.466, -1.714]
  MoveL 4439 to (26.69, 71.11, -199.54) mm, rotated rx -167.81 ry 3.47 rz -52.11 deg; joints [-1.511, -32.037, 98.714, 145.502, 95.313, 28.482, -1.714]
  MoveL 4440 to (27.05, 71.49, -199.54) mm, rotated rx -167.81 ry 3.47 rz -52.11 deg; joints [-1.524, -32.024, 98.679, 145.491, 95.298, 28.499, -1.714]
  MoveL 4441 to (29.29, 73.36, -199.89) mm, rotated rx -167.81 ry 3.47 rz -52.11 deg; joints [-1.611, -31.972, 98.513, 145.42, 95.223, 28.593, -1.714]
  MoveL 4442 to (30.43, 74, -200.32) mm, rotated rx -167.81 ry 3.47 rz -52.11 deg; joints [-1.658, -31.967, 98.467, 145.381, 95.201, 28.631, -1.714]
  MoveL 4443 to (31.57, 74.44, -200.93) mm, rotated rx -167.81 ry 3.47 rz -52.11 deg; joints [-1.706, -31.975, 98.446, 145.34, 95.188, 28.663, -1.714]
  MoveL 4444 to (33.88, 74.73, -202.66) mm, rotated rx -167.81 ry 3.47 rz -52.11 deg; joints [-1.809, -32.032, 98.479, 145.25, 95.191, 28.711, -1.714]
  MoveL 4445 to (36.22, 74.23, -205.08) mm, rotated rx -167.81 ry 3.47 rz -52.11 deg; joints [-1.92, -32.143, 98.61, 145.15, 95.233, 28.737, -1.714]
  MoveL 4446 to (37.98, 73.2, -207.5) mm, rotated rx -167.81 ry 3.47 rz -52.11 deg; joints [-2.01, -32.275, 98.793, 145.068, 95.295, 28.737, -1.714]
  MoveL 4447 to (38.4, 72.58, -208.45) mm, rotated rx -167.81 ry 3.47 rz -52.11 deg; joints [-2.035, -32.335, 98.885, 145.044, 95.327, 28.727, -1.714]
  MoveL 4448 to (38.52, 71.9, -209.23) mm, rotated rx -167.81 ry 3.47 rz -52.11 deg; joints [-2.048, -32.392, 98.979, 145.031, 95.36, 28.71, -1.714]
  MoveL 4449 to (38.47, 71.53, -209.56) mm, rotated rx -167.81 ry 3.47 rz -52.11 deg; joints [-2.049, -32.419, 99.026, 145.028, 95.377, 28.698, -1.714]
  MoveL 4450 to (38.34, 71.15, -209.84) mm, rotated rx -167.81 ry 3.47 rz -52.11 deg; joints [-2.048, -32.445, 99.073, 145.029, 95.394, 28.686, -1.714]
  MoveL 4451 to (37.85, 70.33, -210.27) mm, rotated rx -167.81 ry 3.47 rz -52.11 deg; joints [-2.034, -32.494, 99.168, 145.038, 95.429, 28.655, -1.714]
  MoveL 4452 to (37.07, 69.44, -210.53) mm, rotated rx -167.81 ry 3.47 rz -52.11 deg; joints [-2.008, -32.54, 99.265, 145.058, 95.464, 28.617, -1.714]
  MoveL 4453 to (35.97, 68.49, -210.62) mm, rotated rx -167.81 ry 3.47 rz -52.11 deg; joints [-1.969, -32.582, 99.362, 145.09, 95.501, 28.573, -1.714]
  MoveL 4454 to (35.56, 68.17, -210.62) mm, rotated rx -167.81 ry 3.47 rz -52.11 deg; joints [-1.954, -32.595, 99.394, 145.103, 95.513, 28.557, -1.714]
  MoveL 4455 to (35.19, 67.9, -210.59) mm, rotated rx -167.81 ry 3.47 rz -52.11 deg; joints [-1.94, -32.605, 99.419, 145.114, 95.523, 28.543, -1.714]
  MoveL 4456 to (34.84, 67.66, -210.54) mm, rotated rx -167.81 ry 3.47 rz -52.11 deg; joints [-1.926, -32.613, 99.442, 145.125, 95.531, 28.531, -1.714]
  MoveL 4457 to (34.48, 67.43, -210.48) mm, rotated rx -167.81 ry 3.47 rz -52.11 deg; joints [-1.912, -32.62, 99.462, 145.137, 95.539, 28.519, -1.714]
  MoveL 4458 to (34.11, 67.18, -210.45) mm, rotated rx -167.81 ry 3.47 rz -52.11 deg; joints [-1.898, -32.629, 99.486, 145.149, 95.548, 28.506, -1.714]
  MoveL 4459 to (33.7, 66.87, -210.43) mm, rotated rx -167.81 ry 3.47 rz -52.11 deg; joints [-1.883, -32.641, 99.516, 145.161, 95.559, 28.49, -1.714]
  MoveL 4460 to (33.29, 66.54, -210.43) mm, rotated rx -167.81 ry 3.47 rz -52.11 deg; joints [-1.868, -32.654, 99.548, 145.173, 95.572, 28.475, -1.714]
  MoveL 4461 to (32.9, 66.24, -210.42) mm, rotated rx -167.81 ry 3.47 rz -52.11 deg; joints [-1.853, -32.666, 99.578, 145.185, 95.583, 28.46, -1.714]
  MoveL 4462 to (32.52, 65.95, -210.4) mm, rotated rx -167.81 ry 3.47 rz -52.11 deg; joints [-1.839, -32.677, 99.605, 145.197, 95.593, 28.446, -1.714]
  MoveL 4463 to (32.17, 65.71, -210.35) mm, rotated rx -167.81 ry 3.47 rz -52.11 deg; joints [-1.826, -32.684, 99.627, 145.208, 95.602, 28.433, -1.714]
  MoveL 4464 to (31.82, 65.48, -210.29) mm, rotated rx -167.81 ry 3.47 rz -52.11 deg; joints [-1.812, -32.691, 99.648, 145.22, 95.611, 28.42, -1.714]
  MoveL 4465 to (31.43, 65.21, -210.23) mm, rotated rx -167.81 ry 3.47 rz -52.11 deg; joints [-1.797, -32.699, 99.671, 145.232, 95.62, 28.407, -1.714]
  MoveL 4466 to (30.93, 64.85, -210.2) mm, rotated rx -167.81 ry 3.47 rz -52.11 deg; joints [-1.778, -32.713, 99.706, 145.248, 95.633, 28.389, -1.714]
  MoveL 4467 to (30.3, 64.39, -210.17) mm, rotated rx -167.81 ry 3.47 rz -52.11 deg; joints [-1.755, -32.731, 99.751, 145.267, 95.65, 28.366, -1.714]
  MoveL 4468 to (29.06, 63.41, -210.17) mm, rotated rx -167.81 ry 3.47 rz -52.11 deg; joints [-1.709, -32.77, 99.847, 145.304, 95.686, 28.319, -1.714]
  MoveL 4469 to (28.4, 62.9, -210.14) mm, rotated rx -167.81 ry 3.47 rz -52.11 deg; joints [-1.684, -32.789, 99.895, 145.325, 95.705, 28.294, -1.714]
  MoveL 4470 to (27.9, 62.53, -210.13) mm, rotated rx -167.81 ry 3.47 rz -52.11 deg; joints [-1.665, -32.804, 99.932, 145.34, 95.719, 28.275, -1.714]
  MoveL 4471 to (27.49, 62.26, -210.12) mm, rotated rx -167.81 ry 3.47 rz -52.11 deg; joints [-1.65, -32.816, 99.958, 145.353, 95.727, 28.262, -1.714]
  MoveL 4472 to (27.12, 62.07, -210.1) mm, rotated rx -167.81 ry 3.47 rz -52.11 deg; joints [-1.636, -32.825, 99.978, 145.365, 95.733, 28.252, -1.714]
  MoveL 4473 to (26.92, 62.02, -209.99) mm, rotated rx -167.81 ry 3.47 rz -52.11 deg; joints [-1.628, -32.823, 99.979, 145.372, 95.734, 28.247, -1.714]
  MoveL 4474 to (26.95, 62.08, -209.77) mm, rotated rx -167.81 ry 3.47 rz -52.11 deg; joints [-1.626, -32.807, 99.963, 145.373, 95.733, 28.247, -1.714]
  MoveL 4475 to (27.24, 62.26, -209.43) mm, rotated rx -167.81 ry 3.47 rz -52.11 deg; joints [-1.633, -32.777, 99.927, 145.368, 95.73, 28.252, -1.714]
  MoveL 4476 to (26.59, 62.7, -208.72) mm, rotated rx -167.81 ry 3.47 rz -52.11 deg; joints [-1.602, -32.74, 99.865, 145.397, 95.702, 28.257, -1.714]
  MoveL 4477 to (24.58, 62.58, -208.57) mm, rotated rx -167.81 ry 3.47 rz -52.11 deg; joints [-1.528, -32.773, 99.892, 145.463, 95.682, 28.236, -1.714]
  MoveL 4478 to (22.66, 62.5, -208.29) mm, rotated rx -167.81 ry 3.47 rz -52.11 deg; joints [-1.456, -32.795, 99.909, 145.527, 95.661, 28.216, -1.714]
  MoveL 4479 to (20.73, 62.4, -208.01) mm, rotated rx -167.81 ry 3.47 rz -52.11 deg; joints [-1.383, -32.818, 99.927, 145.592, 95.642, 28.195, -1.714]
  MoveL 4480 to (18.8, 62.29, -207.75) mm, rotated rx -167.81 ry 3.47 rz -52.11 deg; joints [-1.311, -32.841, 99.946, 145.657, 95.622, 28.174, -1.714]
  MoveL 4481 to (16.78, 62.17, -207.53) mm, rotated rx -167.81 ry 3.47 rz -52.11 deg; joints [-1.236, -32.87, 99.97, 145.724, 95.601, 28.152, -1.714]
  MoveL 4482 to (14.66, 62.11, -207.39) mm, rotated rx -167.81 ry 3.47 rz -52.11 deg; joints [-1.158, -32.904, 99.993, 145.794, 95.576, 28.133, -1.714]
  MoveL 4483 to (12.12, 62.14, -207.28) mm, rotated rx -167.81 ry 3.47 rz -52.11 deg; joints [-1.066, -32.947, 100.015, 145.877, 95.538, 28.115, -1.714]
  MoveL 4484 to (9.66, 61.81, -207.2) mm, rotated rx -167.81 ry 3.47 rz -52.11 deg; joints [-0.976, -32.996, 100.067, 145.957, 95.52, 28.085, -1.714]
  MoveL 4485 to (7.56, 61.54, -207.09) mm, rotated rx -167.81 ry 3.47 rz -52.11 deg; joints [-0.899, -33.034, 100.108, 146.025, 95.506, 28.058, -1.714]
  MoveL 4486 to (5.68, 61.34, -206.91) mm, rotated rx -167.81 ry 3.47 rz -52.11 deg; joints [-0.829, -33.063, 100.136, 146.088, 95.49, 28.036, -1.714]
  MoveL 4487 to (3.65, 61.17, -206.79) mm, rotated rx -167.81 ry 3.47 rz -52.11 deg; joints [-0.754, -33.098, 100.167, 146.155, 95.471, 28.014, -1.714]
  MoveL 4488 to (1.57, 61, -206.65) mm, rotated rx -167.81 ry 3.47 rz -52.11 deg; joints [-0.677, -33.133, 100.198, 146.223, 95.451, 27.991, -1.714]
  MoveL 4489 to (-0.6, 60.83, -206.59) mm, rotated rx -167.81 ry 3.47 rz -52.11 deg; joints [-0.598, -33.174, 100.232, 146.293, 95.428, 27.969, -1.714]
  MoveL 4490 to (-2.73, 60.65, -206.36) mm, rotated rx -167.81 ry 3.47 rz -52.11 deg; joints [-0.519, -33.204, 100.259, 146.364, 95.408, 27.945, -1.714]
  MoveL 4491 to (-4.85, 60.47, -206.25) mm, rotated rx -167.81 ry 3.47 rz -52.11 deg; joints [-0.441, -33.24, 100.291, 146.434, 95.387, 27.922, -1.714]
  MoveL 4492 to (-6.98, 60.27, -206.02) mm, rotated rx -167.81 ry 3.47 rz -52.11 deg; joints [-0.361, -33.271, 100.318, 146.505, 95.368, 27.898, -1.714]
  MoveL 4493 to (-9.11, 60.09, -205.91) mm, rotated rx -167.81 ry 3.47 rz -52.11 deg; joints [-0.283, -33.308, 100.35, 146.575, 95.347, 27.875, -1.714]
  MoveL 4494 to (-11.23, 59.89, -205.69) mm, rotated rx -167.81 ry 3.47 rz -52.11 deg; joints [-0.204, -33.338, 100.378, 146.646, 95.327, 27.851, -1.714]
  MoveL 4495 to (-13.36, 59.7, -205.58) mm, rotated rx -167.81 ry 3.47 rz -52.11 deg; joints [-0.126, -33.375, 100.409, 146.715, 95.306, 27.828, -1.714]
  MoveL 4496 to (-15.48, 59.5, -205.48) mm, rotated rx -167.81 ry 3.47 rz -52.11 deg; joints [-0.048, -33.412, 100.441, 146.785, 95.285, 27.806, -1.714]
  MoveL 4497 to (-17.38, 59.27, -205.25) mm, rotated rx -167.81 ry 3.47 rz -52.11 deg; joints [0.024, -33.437, 100.467, 146.849, 95.271, 27.781, -1.714]
  MoveL 4498 to (-19.2, 59.01, -204.95) mm, rotated rx -167.81 ry 3.47 rz -52.11 deg; joints [0.093, -33.457, 100.491, 146.911, 95.26, 27.756, -1.714]
  MoveL 4499 to (-20.97, 58.71, -204.56) mm, rotated rx -167.81 ry 3.47 rz -52.11 deg; joints [0.163, -33.471, 100.514, 146.972, 95.252, 27.729, -1.714]
  MoveL 4500 to (-19.56, 58.54, -203.63) mm, rotated rx -167.81 ry 3.47 rz -52.11 deg; joints [0.123, -33.388, 100.468, 146.935, 95.291, 27.722, -1.714]
  MoveL 4501 to (-19.92, 58.52, -203.58) mm, rotated rx -167.81 ry 3.47 rz -52.11 deg; joints [0.137, -33.392, 100.47, 146.947, 95.287, 27.718, -1.714]
  MoveL 4502 to (-20.3, 58.53, -203.52) mm, rotated rx -167.81 ry 3.47 rz -52.11 deg; joints [0.151, -33.395, 100.471, 146.96, 95.282, 27.715, -1.714]
  MoveL 4503 to (-20.7, 58.62, -203.48) mm, rotated rx -167.81 ry 3.47 rz -52.11 deg; joints [0.166, -33.399, 100.465, 146.973, 95.271, 27.715, -1.714]
  MoveL 4504 to (-21.13, 58.77, -203.46) mm, rotated rx -167.81 ry 3.47 rz -52.11 deg; joints [0.181, -33.404, 100.456, 146.987, 95.256, 27.718, -1.714]
  MoveL 4505 to (-21.58, 58.99, -203.45) mm, rotated rx -167.81 ry 3.47 rz -52.11 deg; joints [0.197, -33.409, 100.442, 147.003, 95.237, 27.723, -1.714]
  MoveL 4506 to (-22.03, 59.23, -203.45) mm, rotated rx -167.81 ry 3.47 rz -52.11 deg; joints [0.212, -33.414, 100.427, 147.017, 95.216, 27.729, -1.714]
  MoveL 4507 to (-22.96, 59.75, -203.45) mm, rotated rx -167.81 ry 3.47 rz -52.11 deg; joints [0.244, -33.424, 100.393, 147.048, 95.173, 27.742, -1.714]
  MoveL 4508 to (-23.39, 59.97, -203.43) mm, rotated rx -167.81 ry 3.47 rz -52.11 deg; joints [0.259, -33.427, 100.378, 147.062, 95.154, 27.747, -1.714]
  MoveL 4509 to (-23.81, 60.17, -203.38) mm, rotated rx -167.81 ry 3.47 rz -52.11 deg; joints [0.274, -33.429, 100.364, 147.077, 95.137, 27.752, -1.714]
  MoveL 4510 to (-24.29, 60.38, -203.3) mm, rotated rx -167.81 ry 3.47 rz -52.11 deg; joints [0.292, -33.43, 100.347, 147.093, 95.119, 27.755, -1.714]
  MoveL 4511 to (-24.81, 60.63, -203.24) mm, rotated rx -167.81 ry 3.47 rz -52.11 deg; joints [0.311, -33.433, 100.329, 147.111, 95.097, 27.76, -1.714]
  MoveL 4512 to (-25.32, 60.89, -203.21) mm, rotated rx -167.81 ry 3.47 rz -52.11 deg; joints [0.329, -33.436, 100.31, 147.128, 95.075, 27.766, -1.714]
  MoveL 4513 to (-25.8, 61.15, -203.19) mm, rotated rx -167.81 ry 3.47 rz -52.11 deg; joints [0.345, -33.441, 100.293, 147.144, 95.053, 27.773, -1.714]
  MoveL 4514 to (-26.27, 61.41, -203.19) mm, rotated rx -167.81 ry 3.47 rz -52.11 deg; joints [0.361, -33.445, 100.276, 147.159, 95.031, 27.779, -1.714]
  MoveL 4515 to (-27.18, 61.92, -203.19) mm, rotated rx -167.81 ry 3.47 rz -52.11 deg; joints [0.392, -33.455, 100.242, 147.189, 94.988, 27.792, -1.714]
  MoveL 4516 to (-28.1, 62.39, -203.17) mm, rotated rx -167.81 ry 3.47 rz -52.11 deg; joints [0.424, -33.464, 100.211, 147.219, 94.948, 27.804, -1.714]
  MoveL 4517 to (-30.38, 63.67, -203.17) mm, rotated rx -167.81 ry 3.47 rz -52.11 deg; joints [0.502, -33.487, 100.127, 147.294, 94.841, 27.836, -1.714]
  MoveL 4518 to (-31.61, 64.44, -203.25) mm, rotated rx -167.81 ry 3.47 rz -52.11 deg; joints [0.543, -33.504, 100.079, 147.333, 94.778, 27.857, -1.714]
  MoveL 4519 to (-32.52, 65.19, -203.52) mm, rotated rx -167.81 ry 3.47 rz -52.11 deg; joints [0.571, -33.527, 100.039, 147.36, 94.719, 27.882, -1.714]
  MoveL 4520 to (-33.12, 65.91, -203.96) mm, rotated rx -167.81 ry 3.47 rz -52.11 deg; joints [0.585, -33.554, 100.007, 147.375, 94.666, 27.909, -1.714]
  MoveL 4521 to (-33.31, 66.26, -204.24) mm, rotated rx -167.81 ry 3.47 rz -52.11 deg; joints [0.587, -33.57, 99.994, 147.379, 94.64, 27.924, -1.714]
  MoveL 4522 to (-33.41, 66.61, -204.57) mm, rotated rx -167.81 ry 3.47 rz -52.11 deg; joints [0.586, -33.587, 99.982, 147.379, 94.616, 27.94, -1.714]
  MoveL 4523 to (-33.39, 67.29, -205.36) mm, rotated rx -167.81 ry 3.47 rz -52.11 deg; joints [0.574, -33.626, 99.965, 147.371, 94.572, 27.975, -1.714]
  MoveL 4524 to (-33.05, 67.95, -206.32) mm, rotated rx -167.81 ry 3.47 rz -52.11 deg; joints [0.549, -33.67, 99.955, 147.351, 94.532, 28.012, -1.714]
  MoveL 4525 to (-31.43, 69.21, -208.78) mm, rotated rx -167.81 ry 3.47 rz -52.11 deg; joints [0.459, -33.774, 99.958, 147.275, 94.467, 28.097, -1.714]
  MoveL 4526 to (-29.15, 70.03, -211.23) mm, rotated rx -167.81 ry 3.47 rz -52.11 deg; joints [0.347, -33.873, 99.99, 147.179, 94.435, 28.172, -1.714]
  MoveL 4527 to (-26.79, 70.09, -212.99) mm, rotated rx -167.81 ry 3.47 rz -52.11 deg; joints [0.243, -33.938, 100.05, 147.086, 94.454, 28.21, -1.714]
  MoveL 4528 to (-25.58, 69.82, -213.6) mm, rotated rx -167.81 ry 3.47 rz -52.11 deg; joints [0.193, -33.957, 100.091, 147.041, 94.483, 28.216, -1.714]
  MoveL 4529 to (-24.35, 69.36, -214.04) mm, rotated rx -167.81 ry 3.47 rz -52.11 deg; joints [0.145, -33.969, 100.139, 146.997, 94.524, 28.212, -1.714]
  MoveL 4530 to (-21.83, 67.87, -214.39) mm, rotated rx -167.81 ry 3.47 rz -52.11 deg; joints [0.055, -33.966, 100.255, 146.912, 94.643, 28.178, -1.714]
  MoveL 4531 to (-19.72, 66.31, -214.39) mm, rotated rx -167.81 ry 3.47 rz -52.11 deg; joints [-0.017, -33.95, 100.363, 146.842, 94.763, 28.134, -1.714]
  MoveL 4532 to (-19.3, 65.99, -214.38) mm, rotated rx -167.81 ry 3.47 rz -52.11 deg; joints [-0.031, -33.946, 100.385, 146.829, 94.787, 28.124, -1.714]
  MoveL 4533 to (-18.88, 65.65, -214.35) mm, rotated rx -167.81 ry 3.47 rz -52.11 deg; joints [-0.045, -33.942, 100.407, 146.815, 94.813, 28.114, -1.714]
  MoveL 4534 to (-18.48, 65.35, -214.34) mm, rotated rx -167.81 ry 3.47 rz -52.11 deg; joints [-0.058, -33.938, 100.427, 146.802, 94.836, 28.106, -1.714]
  MoveL 4535 to (-18.12, 65.1, -214.36) mm, rotated rx -167.81 ry 3.47 rz -52.11 deg; joints [-0.071, -33.936, 100.446, 146.79, 94.855, 28.099, -1.714]
  MoveL 4536 to (-17.71, 64.82, -214.39) mm, rotated rx -167.81 ry 3.47 rz -52.11 deg; joints [-0.085, -33.934, 100.466, 146.776, 94.877, 28.091, -1.714]
  MoveL 4537 to (-17.22, 64.51, -214.45) mm, rotated rx -167.81 ry 3.47 rz -52.11 deg; joints [-0.102, -33.934, 100.49, 146.76, 94.901, 28.084, -1.714]
  MoveL 4538 to (-16.73, 64.21, -214.53) mm, rotated rx -167.81 ry 3.47 rz -52.11 deg; joints [-0.12, -33.934, 100.513, 146.743, 94.924, 28.077, -1.714]
  MoveL 4539 to (-16.25, 63.9, -214.58) mm, rotated rx -167.81 ry 3.47 rz -52.11 deg; joints [-0.137, -33.933, 100.536, 146.727, 94.949, 28.069, -1.714]
  MoveL 4540 to (-15.81, 63.6, -214.6) mm, rotated rx -167.81 ry 3.47 rz -52.11 deg; joints [-0.152, -33.93, 100.558, 146.712, 94.972, 28.061, -1.714]
  MoveL 4541 to (-15.39, 63.3, -214.61) mm, rotated rx -167.81 ry 3.47 rz -52.11 deg; joints [-0.167, -33.927, 100.579, 146.698, 94.995, 28.053, -1.714]
  MoveL 4542 to (-14.97, 62.98, -214.61) mm, rotated rx -167.81 ry 3.47 rz -52.11 deg; joints [-0.181, -33.924, 100.6, 146.684, 95.019, 28.044, -1.714]
  MoveL 4543 to (-14.5, 62.67, -214.65) mm, rotated rx -167.81 ry 3.47 rz -52.11 deg; joints [-0.198, -33.922, 100.623, 146.668, 95.043, 28.036, -1.714]
  MoveL 4544 to (-14.03, 62.38, -214.7) mm, rotated rx -167.81 ry 3.47 rz -52.11 deg; joints [-0.214, -33.921, 100.645, 146.652, 95.066, 28.028, -1.714]
  MoveL 4545 to (-13.55, 62.1, -214.77) mm, rotated rx -167.81 ry 3.47 rz -52.11 deg; joints [-0.232, -33.92, 100.666, 146.635, 95.088, 28.022, -1.714]
  MoveL 4546 to (-13.09, 61.9, -214.83) mm, rotated rx -167.81 ry 3.47 rz -52.11 deg; joints [-0.249, -33.918, 100.681, 146.62, 95.106, 28.018, -1.714]
  MoveL 4547 to (-12.65, 61.75, -214.86) mm, rotated rx -167.81 ry 3.47 rz -52.11 deg; joints [-0.264, -33.913, 100.69, 146.605, 95.121, 28.016, -1.714]
  MoveL 4548 to (-12.25, 61.68, -214.87) mm, rotated rx -167.81 ry 3.47 rz -52.11 deg; joints [-0.279, -33.907, 100.692, 146.592, 95.131, 28.016, -1.714]
  MoveL 4549 to (-11.86, 61.65, -214.87) mm, rotated rx -167.81 ry 3.47 rz -52.11 deg; joints [-0.293, -33.9, 100.691, 146.579, 95.138, 28.018, -1.714]
  MoveL 4550 to (-13.12, 61.93, -215.74) mm, rotated rx -167.81 ry 3.47 rz -52.11 deg; joints [-0.258, -33.976, 100.724, 146.612, 95.096, 28.03, -1.714]
  MoveL 4551 to (-11.52, 61.97, -216.02) mm, rotated rx -167.81 ry 3.47 rz -52.11 deg; joints [-0.319, -33.962, 100.717, 146.557, 95.115, 28.046, -1.714]
  MoveL 4552 to (-9.72, 61.96, -216.22) mm, rotated rx -167.81 ry 3.47 rz -52.11 deg; joints [-0.386, -33.939, 100.709, 146.497, 95.142, 28.06, -1.714]
  MoveL 4553 to (-7.67, 61.92, -216.35) mm, rotated rx -167.81 ry 3.47 rz -52.11 deg; joints [-0.461, -33.908, 100.698, 146.429, 95.175, 28.074, -1.714]
  MoveL 4554 to (-5.42, 61.83, -216.44) mm, rotated rx -167.81 ry 3.47 rz -52.11 deg; joints [-0.543, -33.871, 100.686, 146.355, 95.213, 28.087, -1.714]
  MoveL 4555 to (-3.28, 61.77, -216.59) mm, rotated rx -167.81 ry 3.47 rz -52.11 deg; joints [-0.621, -33.84, 100.675, 146.284, 95.248, 28.101, -1.714]
  MoveL 4556 to (-1.15, 61.71, -216.8) mm, rotated rx -167.81 ry 3.47 rz -52.11 deg; joints [-0.701, -33.812, 100.667, 146.213, 95.281, 28.116, -1.714]
  MoveL 4557 to (0.88, 61.65, -216.92) mm, rotated rx -167.81 ry 3.47 rz -52.11 deg; joints [-0.775, -33.781, 100.656, 146.146, 95.314, 28.129, -1.714]
  MoveL 4558 to (2.73, 61.61, -217.19) mm, rotated rx -167.81 ry 3.47 rz -52.11 deg; joints [-0.844, -33.762, 100.652, 146.083, 95.342, 28.144, -1.714]
  MoveL 4559 to (4.79, 61.55, -217.4) mm, rotated rx -167.81 ry 3.47 rz -52.11 deg; joints [-0.921, -33.736, 100.645, 146.014, 95.374, 28.158, -1.714]
  MoveL 4560 to (6.87, 61.47, -217.54) mm, rotated rx -167.81 ry 3.47 rz -52.11 deg; joints [-0.997, -33.705, 100.635, 145.945, 95.408, 28.171, -1.714]
  MoveL 4561 to (9.01, 61.38, -217.65) mm, rotated rx -167.81 ry 3.47 rz -52.11 deg; joints [-1.075, -33.67, 100.623, 145.875, 95.444, 28.184, -1.714]
  MoveL 4562 to (11.13, 61.3, -217.88) mm, rotated rx -167.81 ry 3.47 rz -52.11 deg; joints [-1.154, -33.644, 100.616, 145.804, 95.478, 28.198, -1.714]
  MoveL 4563 to (13.27, 61.19, -218.14) mm, rotated rx -167.81 ry 3.47 rz -52.11 deg; joints [-1.234, -33.619, 100.612, 145.732, 95.513, 28.212, -1.714]
  MoveL 4564 to (15.39, 61.09, -218.23) mm, rotated rx -167.81 ry 3.47 rz -52.11 deg; joints [-1.311, -33.584, 100.6, 145.662, 95.549, 28.224, -1.714]
  MoveL 4565 to (17.57, 60.99, -218.27) mm, rotated rx -167.81 ry 3.47 rz -52.11 deg; joints [-1.389, -33.544, 100.584, 145.591, 95.585, 28.236, -1.714]
  MoveL 4566 to (19.68, 60.89, -218.37) mm, rotated rx -167.81 ry 3.47 rz -52.11 deg; joints [-1.466, -33.51, 100.572, 145.521, 95.621, 28.248, -1.714]
  MoveL 4567 to (21.8, 60.77, -218.58) mm, rotated rx -167.81 ry 3.47 rz -52.11 deg; joints [-1.544, -33.482, 100.565, 145.45, 95.656, 28.262, -1.714]
  MoveL 4568 to (23.87, 60.65, -218.91) mm, rotated rx -167.81 ry 3.47 rz -52.11 deg; joints [-1.623, -33.463, 100.566, 145.38, 95.689, 28.275, -1.714]
  MoveL 4569 to (26.02, 60.5, -219.17) mm, rotated rx -167.81 ry 3.47 rz -52.11 deg; joints [-1.703, -33.438, 100.564, 145.307, 95.726, 28.288, -1.714]
  MoveL 4570 to (28.15, 60.36, -219.37) mm, rotated rx -167.81 ry 3.47 rz -52.11 deg; joints [-1.781, -33.409, 100.559, 145.236, 95.762, 28.3, -1.714]
